LIN {X 0,Y 382.993,Z 296.779,A -85,B 0,C 180,E1 -12093.4,E2 -12093.4} C_VEL
LIN {X 0,Y 383.024,Z 296.771,A -85,B 0,C 180,E1 -12096.162,E2 -12096.162} C_VEL
LIN {X 0,Y 382.969,Z 296.778,A -85,B 0,C 180,E1 -12099.961,E2 -12099.961} C_VEL
LIN {X 0,Y 382.998,Z 296.778,A -85,B 0,C 180,E1 -12102.777,E2 -12102.777} C_VEL
LIN {X 0,Y 382.989,Z 296.776,A -85,B 0,C 180,E1 -12105.788,E2 -12105.788} C_VEL
LIN {X 0,Y 382.981,Z 296.782,A -85,B 0,C 180,E1 -12108.794,E2 -12108.794} C_VEL
LIN {X 0,Y 382.993,Z 296.776,A -85,B 0,C 180,E1 -12112.095,E2 -12112.095} C_VEL
LIN {X 0,Y 383.009,Z 296.776,A -85,B 0,C 180,E1 -12115.331,E2 -12115.331} C_VEL
LIN {X 0,Y 382.978,Z 296.781,A -85,B 0,C 180,E1 -12119.081,E2 -12119.081} C_VEL
LIN {X 0,Y 383.046,Z 296.772,A -85,B 0,C 180,E1 -12122.697,E2 -12122.697} C_VEL
LIN {X 0,Y 383.041,Z 296.772,A -85,B 0,C 180,E1 -12125.039,E2 -12125.039} C_VEL
LIN {X 0,Y 382.982,Z 296.78,A -85,B 0,C 180,E1 -12128.468,E2 -12128.468} C_VEL
LIN {X 0,Y 383.078,Z 296.767,A -85,B 0,C 180,E1 -12131.827,E2 -12131.827} C_VEL
LIN {X 0,Y 383.098,Z 296.763,A -85,B 0,C 180,E1 -12135.118,E2 -12135.118} C_VEL
LIN {X 0,Y 383.085,Z 296.769,A -85,B 0,C 180,E1 -12138.357,E2 -12138.357} C_VEL
LIN {X 0,Y 383.202,Z 296.753,A -85,B 0,C 180,E1 -12142.028,E2 -12142.028} C_VEL
LIN {X 0,Y 383.168,Z 296.754,A -85,B 0,C 180,E1 -12144.738,E2 -12144.738} C_VEL
LIN {X 0,Y 383.361,Z 296.733,A -85,B 0,C 180,E1 -12147.899,E2 -12147.899} C_VEL
LIN {X 0,Y 383.246,Z 296.743,A -85,B 0,C 180,E1 -12151.051,E2 -12151.051} C_VEL
LIN {X 0,Y 383.361,Z 296.733,A -85,B 0,C 180,E1 -12152.101,E2 -12152.101} C_VEL
LIN {X 0,Y 383.23,Z 296.747,A -85,B 0,C 180,E1 -12156.317,E2 -12156.317} C_VEL
LIN {X 0,Y 383.131,Z 296.762,A -85,B 0,C 180,E1 -12159.503,E2 -12159.503} C_VEL
LIN {X 0,Y 383.113,Z 296.766,A -85,B 0,C 180,E1 -12163.537,E2 -12163.537} C_VEL
LIN {X 0,Y 383.083,Z 296.769,A -85,B 0,C 180,E1 -12167.455,E2 -12167.455} C_VEL
LIN {X 0,Y 383.017,Z 296.773,A -85,B 0,C 180,E1 -12170.648,E2 -12170.648} C_VEL
LIN {X 0,Y 383.022,Z 296.775,A -85,B 0,C 180,E1 -12173.808,E2 -12173.808} C_VEL
LIN {X 0,Y 383.069,Z 296.767,A -85,B 0,C 180,E1 -12176.124,E2 -12176.124} C_VEL
LIN {X 0,Y 383.039,Z 296.771,A -85,B 0,C 180,E1 -12178.493,E2 -12178.493} C_VEL
LIN {X 0,Y 383.003,Z 296.775,A -85,B 0,C 180,E1 -12182.15,E2 -12182.15} C_VEL
LIN {X 0,Y 383.007,Z 296.775,A -85,B 0,C 180,E1 -12184.534,E2 -12184.534} C_VEL
LIN {X 0,Y 382.344,Z 296.861,A -85,B 0,C 180,E1 -12185.411,E2 -12185.411} C_VEL
LIN {X 0,Y 379.471,Z 297.217,A -85,B 0,C 180,E1 -12186.835,E2 -12186.835} C_VEL
LIN {X 0,Y 377.045,Z 297.517,A -85,B 0,C 180,E1 -12187.987,E2 -12187.987} C_VEL
LIN {X 0,Y 376.019,Z 297.647,A -85,B 0,C 180,E1 -12188.878,E2 -12188.878} C_VEL
LIN {X 0,Y 375.944,Z 297.654,A -85,B 0,C 180,E1 -12189.18,E2 -12189.18} C_VEL
LIN {X 0,Y 375.924,Z 297.657,A -85,B 0,C 180,E1 -12192.302,E2 -12192.302} C_VEL
LIN {X 0,Y 375.919,Z 297.66,A -85,B 0,C 180,E1 -12195.27,E2 -12195.27} C_VEL
LIN {X 0,Y 375.911,Z 297.659,A -85,B 0,C 180,E1 -12198.404,E2 -12198.404} C_VEL
LIN {X 0,Y 375.947,Z 297.652,A -85,B 0,C 180,E1 -12201.912,E2 -12201.912} C_VEL
LIN {X 0,Y 375.973,Z 297.65,A -85,B 0,C 180,E1 -12205.335,E2 -12205.335} C_VEL
LIN {X 0,Y 376.132,Z 297.715,A -85,B 0,C 180,E1 -12208.895,E2 -12208.895} C_VEL
LIN {X 0,Y 376.163,Z 302.091,A -85,B 0,C 180,E1 -12211.417,E2 -12211.417} C_VEL
LIN {X 0,Y 375.789,Z 308.656,A -85,B 0,C 180,E1 -12215.117,E2 -12215.117} C_VEL
LIN {X 0,Y 375.538,Z 314.97,A -85,B 0,C 180,E1 -12218.598,E2 -12218.598} C_VEL
LIN {X 0,Y 375.35,Z 320.211,A -85,B 0,C 180,E1 -12221.441,E2 -12221.441} C_VEL
LIN {X 0,Y 375.145,Z 326.489,A -85,B 0,C 180,E1 -12224.796,E2 -12224.796} C_VEL
LIN {X 0,Y 375.052,Z 332.791,A -85,B 0,C 180,E1 -12228.106,E2 -12228.106} C_VEL
LIN {X 0,Y 375.004,Z 334.24,A -85,B 0,C 180,E1 -12228.858,E2 -12228.858} C_VEL
LIN {X 0,Y 376.479,Z 346.042,A -85,B 0,C 180,E1 -12229.583,E2 -12229.583} C_VEL
LIN {X 0,Y 376.877,Z 352.36,A -85,B 0,C 180,E1 -12230.069,E2 -12230.069} C_VEL
LIN {X 0,Y 376.461,Z 362.339,A -85,B 0,C 180,E1 -12231.006,E2 -12231.006} C_VEL
LIN {X 0,Y 376.1,Z 370.955,A -85,B 0,C 180,E1 -12232.05,E2 -12232.05} C_VEL
LIN {X 0,Y 375.834,Z 378.97,A -85,B 0,C 180,E1 -12233.29,E2 -12233.29} C_VEL
LIN {X 0,Y 375.594,Z 385.708,A -85,B 0,C 180,E1 -12234.633,E2 -12234.633} C_VEL
LIN {X 0,Y 375.366,Z 389.937,A -85,B 0,C 180,E1 -12235.706,E2 -12235.706} C_VEL
LIN {X 0,Y 375.173,Z 393.311,A -85,B 0,C 180,E1 -12236.78,E2 -12236.78} C_VEL
LIN {X 0,Y 375.035,Z 395.913,A -85,B 0,C 180,E1 -12237.854,E2 -12237.854} C_VEL
LIN {X 0,Y 374.985,Z 397.794,A -85,B 0,C 180,E1 -12238.928,E2 -12238.928} C_VEL
LIN {X 0,Y 374.972,Z 398.993,A -85,B 0,C 180,E1 -12240.001,E2 -12240.001} C_VEL
LIN {X 0,Y 375.035,Z 399.523,A -85,B 0,C 180,E1 -12241.075,E2 -12241.075} C_VEL
LIN {X 0,Y 375.176,Z 399.397,A -85,B 0,C 180,E1 -12242.148,E2 -12242.148} C_VEL
LIN {X 0,Y 375.419,Z 398.616,A -85,B 0,C 180,E1 -12243.221,E2 -12243.221} C_VEL
LIN {X 0,Y 376.126,Z 396.159,A -85,B 0,C 180,E1 -12244.825,E2 -12244.825} C_VEL
LIN {X 0,Y 376.703,Z 392.135,A -85,B 0,C 180,E1 -12246.428,E2 -12246.428} C_VEL
LIN {X 0,Y 377.569,Z 386.275,A -85,B 0,C 180,E1 -12248.026,E2 -12248.026} C_VEL
LIN {X 0,Y 378.359,Z 379.801,A -85,B 0,C 180,E1 -12249.355,E2 -12249.355} C_VEL
LIN {X 0,Y 379.334,Z 372.3,A -85,B 0,C 180,E1 -12250.549,E2 -12250.549} C_VEL
LIN {X 0,Y 380.313,Z 362.823,A -85,B 0,C 180,E1 -12251.73,E2 -12251.73} C_VEL
LIN {X 0,Y 380.625,Z 357.706,A -85,B 0,C 180,E1 -12252.261,E2 -12252.261} C_VEL
LIN {X 0,Y 379.01,Z 348.75,A -85,B 0,C 180,E1 -12253.193,E2 -12253.193} C_VEL
LIN {X 0,Y 376.292,Z 338.883,A -85,B 0,C 180,E1 -12254.122,E2 -12254.122} C_VEL
LIN {X 0,Y 376.791,Z 332.831,A -85,B 0,C 180,E1 -12257.96,E2 -12257.96} C_VEL
LIN {X 0,Y 377.374,Z 327.03,A -85,B 0,C 180,E1 -12261.869,E2 -12261.869} C_VEL
LIN {X 0,Y 377.99,Z 322.325,A -85,B 0,C 180,E1 -12265.319,E2 -12265.319} C_VEL
LIN {X 0,Y 378.845,Z 317.93,A -85,B 0,C 180,E1 -12268.839,E2 -12268.839} C_VEL
LIN {X 0,Y 379.207,Z 315.14,A -85,B 0,C 180,E1 -12271.511,E2 -12271.511} C_VEL
LIN {X 0,Y 379.155,Z 313.11,A -85,B 0,C 180,E1 -12273.786,E2 -12273.786} C_VEL
LIN {X 0,Y 379.022,Z 311.404,A -85,B 0,C 180,E1 -12276.397,E2 -12276.397} C_VEL
LIN {X 0,Y 378.859,Z 310.258,A -85,B 0,C 180,E1 -12279.104,E2 -12279.104} C_VEL
LIN {X 0,Y 378.886,Z 309.796,A -85,B 0,C 180,E1 -12282.101,E2 -12282.101} C_VEL
LIN {X 0,Y 379.077,Z 310.446,A -85,B 0,C 180,E1 -12285.21,E2 -12285.21} C_VEL
LIN {X 0,Y 379.596,Z 312.145,A -85,B 0,C 180,E1 -12288.201,E2 -12288.201} C_VEL
LIN {X 0,Y 380.322,Z 314.889,A -85,B 0,C 180,E1 -12291.076,E2 -12291.076} C_VEL
LIN {X 0,Y 381.298,Z 319.139,A -85,B 0,C 180,E1 -12294.195,E2 -12294.195} C_VEL
LIN {X 0,Y 382.493,Z 324.452,A -85,B 0,C 180,E1 -12297.178,E2 -12297.178} C_VEL
LIN {X 0,Y 383.114,Z 328.518,A -85,B 0,C 180,E1 -12299.093,E2 -12299.093} C_VEL
LIN {X 0,Y 382.773,Z 331.551,A -85,B 0,C 180,E1 -12300.281,E2 -12300.281} C_VEL
LIN {X 0,Y 380.4,Z 341.516,A -85,B 0,C 180,E1 -12303.678,E2 -12303.678} C_VEL
LIN {X 0,Y 378.337,Z 354.145,A -85,B 0,C 180,E1 -12307.616,E2 -12307.616} C_VEL
LIN {X 0,Y 377.129,Z 364.425,A -85,B 0,C 180,E1 -12310.537,E2 -12310.537} C_VEL
LIN {X 0,Y 379.386,Z 377.001,A -85,B 0,C 180,E1 -12311.197,E2 -12311.197} C_VEL
LIN {X 0,Y 380.292,Z 388.82,A -85,B 0,C 180,E1 -12311.915,E2 -12311.915} C_VEL
LIN {X 0,Y 380.196,Z 399.286,A -85,B 0,C 180,E1 -12312.67,E2 -12312.67} C_VEL
LIN {X 0,Y 379.013,Z 411.289,A -85,B 0,C 180,E1 -12313.712,E2 -12313.712} C_VEL
LIN {X 0,Y 377.852,Z 422.147,A -85,B 0,C 180,E1 -12314.906,E2 -12314.906} C_VEL
LIN {X 0,Y 376.925,Z 431.899,A -85,B 0,C 180,E1 -12316.247,E2 -12316.247} C_VEL
LIN {X 0,Y 376.109,Z 439.941,A -85,B 0,C 180,E1 -12317.591,E2 -12317.591} C_VEL
LIN {X 0,Y 375.361,Z 447.84,A -85,B 0,C 180,E1 -12319.209,E2 -12319.209} C_VEL
LIN {X 0,Y 374.984,Z 454.183,A -85,B 0,C 180,E1 -12320.833,E2 -12320.833} C_VEL
LIN {X 0,Y 374.858,Z 459.235,A -85,B 0,C 180,E1 -12322.459,E2 -12322.459} C_VEL
LIN {X 0,Y 374.782,Z 462.239,A -85,B 0,C 180,E1 -12323.659,E2 -12323.659} C_VEL
LIN {X 0,Y 374.773,Z 464.187,A -85,B 0,C 180,E1 -12324.62,E2 -12324.62} C_VEL
LIN {X 0,Y 374.759,Z 465.952,A -85,B 0,C 180,E1 -12325.698,E2 -12325.698} C_VEL
LIN {X 0,Y 374.922,Z 467.299,A -85,B 0,C 180,E1 -12326.776,E2 -12326.776} C_VEL
LIN {X 0,Y 374.99,Z 468.16,A -85,B 0,C 180,E1 -12327.852,E2 -12327.852} C_VEL
LIN {X 0,Y 374.931,Z 468.593,A -85,B 0,C 180,E1 -12328.926,E2 -12328.926} C_VEL
LIN {X 0,Y 374.902,Z 468.611,A -85,B 0,C 180,E1 -12330,E2 -12330} C_VEL
LIN {X 0,Y 374.93,Z 468.155,A -85,B 0,C 180,E1 -12331.074,E2 -12331.074} C_VEL
LIN {X 0,Y 375.039,Z 467.282,A -85,B 0,C 180,E1 -12332.148,E2 -12332.148} C_VEL
LIN {X 0,Y 374.995,Z 465.962,A -85,B 0,C 180,E1 -12333.223,E2 -12333.223} C_VEL
LIN {X 0,Y 374.841,Z 463.042,A -85,B 0,C 180,E1 -12334.84,E2 -12334.84} C_VEL
LIN {X 0,Y 374.949,Z 458.664,A -85,B 0,C 180,E1 -12336.567,E2 -12336.567} C_VEL
LIN {X 0,Y 374.995,Z 452.62,A -85,B 0,C 180,E1 -12338.352,E2 -12338.352} C_VEL
LIN {X 0,Y 375.182,Z 445.526,A -85,B 0,C 180,E1 -12339.978,E2 -12339.978} C_VEL
LIN {X 0,Y 375.676,Z 436.584,A -85,B 0,C 180,E1 -12341.602,E2 -12341.602} C_VEL
LIN {X 0,Y 376.261,Z 427.274,A -85,B 0,C 180,E1 -12342.953,E2 -12342.953} C_VEL
LIN {X 0,Y 376.815,Z 416.818,A -85,B 0,C 180,E1 -12344.17,E2 -12344.17} C_VEL
LIN {X 0,Y 377.38,Z 406.757,A -85,B 0,C 180,E1 -12345.113,E2 -12345.113} C_VEL
LIN {X 0,Y 378.045,Z 394.838,A -85,B 0,C 180,E1 -12345.984,E2 -12345.984} C_VEL
LIN {X 0,Y 377.323,Z 383.251,A -85,B 0,C 180,E1 -12346.641,E2 -12346.641} C_VEL
LIN {X 0,Y 376.34,Z 371.136,A -85,B 0,C 180,E1 -12347.14,E2 -12347.14} C_VEL
LIN {X 0,Y 376.014,Z 366.072,A -85,B 0,C 180,E1 -12347.296,E2 -12347.296} C_VEL
LIN {X 0,Y 377.114,Z 351.417,A -85,B 0,C 180,E1 -12351.278,E2 -12351.278} C_VEL
LIN {X 0,Y 378.263,Z 339.903,A -85,B 0,C 180,E1 -12354.437,E2 -12354.437} C_VEL
LIN {X 0,Y 379.811,Z 327.577,A -85,B 0,C 180,E1 -12357.854,E2 -12357.854} C_VEL
LIN {X 0,Y 380.623,Z 320.323,A -85,B 0,C 180,E1 -12359.904,E2 -12359.904} C_VEL
LIN {X 0,Y 378.647,Z 310.587,A -85,B 0,C 180,E1 -12362.917,E2 -12362.917} C_VEL
LIN {X 0,Y 376.227,Z 298.875,A -85,B 0,C 180,E1 -12366.71,E2 -12366.71} C_VEL
LIN {X 0,Y 375.972,Z 297.654,A -85,B 0,C 180,E1 -12367.158,E2 -12367.158} C_VEL
LIN {X 0,Y 375.945,Z 297.656,A -85,B 0,C 180,E1 -12370.867,E2 -12370.867} C_VEL
LIN {X 0,Y 375.935,Z 297.658,A -85,B 0,C 180,E1 -12373.765,E2 -12373.765} C_VEL
LIN {X 0,Y 375.939,Z 297.655,A -85,B 0,C 180,E1 -12376.81,E2 -12376.81} C_VEL
LIN {X 0,Y 375.968,Z 297.655,A -85,B 0,C 180,E1 -12380.537,E2 -12380.537} C_VEL
LIN {X 0,Y 375.969,Z 297.655,A -85,B 0,C 180,E1 -12383.495,E2 -12383.495} C_VEL
LIN {X 0,Y 375.969,Z 297.686,A -85,B 0,C 180,E1 -12385.888,E2 -12385.888} C_VEL
LIN {X 0,Y 377.371,Z 303.877,A -85,B 0,C 180,E1 -12388.947,E2 -12388.947} C_VEL
LIN {X 0,Y 377.839,Z 308.436,A -85,B 0,C 180,E1 -12391.077,E2 -12391.077} C_VEL
LIN {X 0,Y 377.468,Z 316.369,A -85,B 0,C 180,E1 -12394.643,E2 -12394.643} C_VEL
LIN {X 0,Y 377.21,Z 324.059,A -85,B 0,C 180,E1 -12398.121,E2 -12398.121} C_VEL
LIN {X 0,Y 376.985,Z 331.514,A -85,B 0,C 180,E1 -12401.522,E2 -12401.522} C_VEL
LIN {X 0,Y 376.762,Z 338.786,A -85,B 0,C 180,E1 -12404.86,E2 -12404.86} C_VEL
LIN {X 0,Y 376.729,Z 345.225,A -85,B 0,C 180,E1 -12407.764,E2 -12407.764} C_VEL
LIN {X 0,Y 379.03,Z 354.751,A -85,B 0,C 180,E1 -12408.501,E2 -12408.501} C_VEL
LIN {X 0,Y 379.112,Z 359.76,A -85,B 0,C 180,E1 -12408.91,E2 -12408.91} C_VEL
LIN {X 0,Y 378.621,Z 367.683,A -85,B 0,C 180,E1 -12409.672,E2 -12409.672} C_VEL
LIN {X 0,Y 377.863,Z 375.923,A -85,B 0,C 180,E1 -12410.705,E2 -12410.705} C_VEL
LIN {X 0,Y 377.418,Z 382.05,A -85,B 0,C 180,E1 -12411.701,E2 -12411.701} C_VEL
LIN {X 0,Y 376.994,Z 387.186,A -85,B 0,C 180,E1 -12412.77,E2 -12412.77} C_VEL
LIN {X 0,Y 376.468,Z 392.079,A -85,B 0,C 180,E1 -12414.105,E2 -12414.105} C_VEL
LIN {X 0,Y 376.109,Z 394.999,A -85,B 0,C 180,E1 -12415.175,E2 -12415.175} C_VEL
LIN {X 0,Y 375.379,Z 397.85,A -85,B 0,C 180,E1 -12416.779,E2 -12416.779} C_VEL
LIN {X 0,Y 375.142,Z 398.857,A -85,B 0,C 180,E1 -12417.851,E2 -12417.851} C_VEL
LIN {X 0,Y 375.01,Z 399.169,A -85,B 0,C 180,E1 -12418.925,E2 -12418.925} C_VEL
LIN {X 0,Y 374.955,Z 398.796,A -85,B 0,C 180,E1 -12419.999,E2 -12419.999} C_VEL
LIN {X 0,Y 374.976,Z 397.723,A -85,B 0,C 180,E1 -12421.073,E2 -12421.073} C_VEL
LIN {X 0,Y 375.035,Z 395.927,A -85,B 0,C 180,E1 -12422.146,E2 -12422.146} C_VEL
LIN {X 0,Y 375.309,Z 391.751,A -85,B 0,C 180,E1 -12423.756,E2 -12423.756} C_VEL
LIN {X 0,Y 375.545,Z 386.75,A -85,B 0,C 180,E1 -12425.098,E2 -12425.098} C_VEL
LIN {X 0,Y 375.658,Z 381.546,A -85,B 0,C 180,E1 -12426.174,E2 -12426.174} C_VEL
LIN {X 0,Y 375.825,Z 374.325,A -85,B 0,C 180,E1 -12427.337,E2 -12427.337} C_VEL
LIN {X 0,Y 376.022,Z 366.64,A -85,B 0,C 180,E1 -12428.3,E2 -12428.3} C_VEL
LIN {X 0,Y 376.267,Z 357.879,A -85,B 0,C 180,E1 -12429.134,E2 -12429.134} C_VEL
LIN {X 0,Y 376.381,Z 348.482,A -85,B 0,C 180,E1 -12429.809,E2 -12429.809} C_VEL
LIN {X 0,Y 375.44,Z 341.359,A -85,B 0,C 180,E1 -12430.208,E2 -12430.208} C_VEL
LIN {X 0,Y 375.56,Z 334.224,A -85,B 0,C 180,E1 -12433.319,E2 -12433.319} C_VEL
LIN {X 0,Y 375.568,Z 325.063,A -85,B 0,C 180,E1 -12437.376,E2 -12437.376} C_VEL
LIN {X 0,Y 375.686,Z 317.354,A -85,B 0,C 180,E1 -12440.818,E2 -12440.818} C_VEL
LIN {X 0,Y 375.83,Z 309.622,A -85,B 0,C 180,E1 -12444.291,E2 -12444.291} C_VEL
LIN {X 0,Y 375.918,Z 303.002,A -85,B 0,C 180,E1 -12447.259,E2 -12447.259} C_VEL
LIN {X 0,Y 376.07,Z 297.64,A -85,B 0,C 180,E1 -12449.683,E2 -12449.683} C_VEL
LIN {X 0,Y 375.942,Z 297.655,A -85,B 0,C 180,E1 -12452.827,E2 -12452.827} C_VEL
LIN {X 0,Y 375.95,Z 297.656,A -85,B 0,C 180,E1 -12455.414,E2 -12455.414} C_VEL
LIN {X 0,Y 375.93,Z 297.655,A -85,B 0,C 180,E1 -12458.262,E2 -12458.262} C_VEL
LIN {X 0,Y 375.912,Z 297.659,A -85,B 0,C 180,E1 -12461.597,E2 -12461.597} C_VEL
LIN {X 0,Y 375.919,Z 297.66,A -85,B 0,C 180,E1 -12464.73,E2 -12464.73} C_VEL
LIN {X 0,Y 375.927,Z 297.657,A -85,B 0,C 180,E1 -12468.398,E2 -12468.398} C_VEL
LIN {X 0,Y 375.968,Z 297.651,A -85,B 0,C 180,E1 -12471.728,E2 -12471.728} C_VEL
LIN {X 0,Y 375.971,Z 297.652,A -85,B 0,C 180,E1 -12475.331,E2 -12475.331} C_VEL
LIN {X 0,Y 375.952,Z 297.657,A -85,B 0,C 180,E1 -12478.437,E2 -12478.437} C_VEL
LIN {X 0,Y 375.992,Z 297.65,A -85,B 0,C 180,E1 -12482.141,E2 -12482.141} C_VEL
LIN {X 0,Y 375.996,Z 297.651,A -85,B 0,C 180,E1 -12484.538,E2 -12484.538} C_VEL
LIN {X 0,Y 375.952,Z 297.655,A -85,B 0,C 180,E1 -12488.045,E2 -12488.045} C_VEL
LIN {X 0,Y 376.012,Z 297.645,A -85,B 0,C 180,E1 -12491.473,E2 -12491.473} C_VEL
LIN {X 0,Y 376.046,Z 297.643,A -85,B 0,C 180,E1 -12494.832,E2 -12494.832} C_VEL
LIN {X 0,Y 376.037,Z 297.645,A -85,B 0,C 180,E1 -12498.136,E2 -12498.136} C_VEL
LIN {X 0,Y 376.174,Z 297.628,A -85,B 0,C 180,E1 -12501.953,E2 -12501.953} C_VEL
LIN {X 0,Y 376.139,Z 297.63,A -85,B 0,C 180,E1 -12504.639,E2 -12504.639} C_VEL
LIN {X 0,Y 376.325,Z 297.609,A -85,B 0,C 180,E1 -12507.859,E2 -12507.859} C_VEL
LIN {X 0,Y 376.218,Z 297.618,A -85,B 0,C 180,E1 -12511.07,E2 -12511.07} C_VEL
LIN {X 0,Y 376.326,Z 297.609,A -85,B 0,C 180,E1 -12512.141,E2 -12512.141} C_VEL
LIN {X 0,Y 376.189,Z 297.624,A -85,B 0,C 180,E1 -12516.436,E2 -12516.436} C_VEL
LIN {X 0,Y 376.101,Z 297.639,A -85,B 0,C 180,E1 -12519.682,E2 -12519.682} C_VEL
LIN {X 0,Y 376.077,Z 297.641,A -85,B 0,C 180,E1 -12523.658,E2 -12523.658} C_VEL
LIN {X 0,Y 376.033,Z 297.646,A -85,B 0,C 180,E1 -12527.608,E2 -12527.608} C_VEL
LIN {X 0,Y 375.967,Z 297.652,A -85,B 0,C 180,E1 -12530.833,E2 -12530.833} C_VEL
LIN {X 0,Y 375.983,Z 297.649,A -85,B 0,C 180,E1 -12534.282,E2 -12534.282} C_VEL
LIN {X 0,Y 376.009,Z 297.646,A -85,B 0,C 180,E1 -12536.653,E2 -12536.653} C_VEL
LIN {X 0,Y 375.967,Z 297.655,A -85,B 0,C 180,E1 -12539.08,E2 -12539.08} C_VEL
LIN {X 0,Y 375.941,Z 297.657,A -85,B 0,C 180,E1 -12542.83,E2 -12542.83} C_VEL
LIN {X 0,Y 375.949,Z 297.657,A -85,B 0,C 180,E1 -12545.417,E2 -12545.417} C_VEL
LIN {X 0,Y 375.944,Z 297.654,A -85,B 0,C 180,E1 -12549.18,E2 -12549.18} C_VEL
LIN {X 0,Y 375.299,Z 297.739,A -85,B 0,C 180,E1 -12550.074,E2 -12550.074} C_VEL
LIN {X 0,Y 372.447,Z 298.096,A -85,B 0,C 180,E1 -12551.527,E2 -12551.527} C_VEL
LIN {X 0,Y 370.01,Z 298.396,A -85,B 0,C 180,E1 -12552.702,E2 -12552.702} C_VEL
LIN {X 0,Y 368.951,Z 298.526,A -85,B 0,C 180,E1 -12553.611,E2 -12553.611} C_VEL
LIN {X 0,Y 368.859,Z 298.536,A -85,B 0,C 180,E1 -12553.919,E2 -12553.919} C_VEL
LIN {X 0,Y 368.878,Z 298.536,A -85,B 0,C 180,E1 -12556.697,E2 -12556.697} C_VEL
LIN {X 0,Y 368.877,Z 298.534,A -85,B 0,C 180,E1 -12559.65,E2 -12559.65} C_VEL
LIN {X 0,Y 368.893,Z 298.534,A -85,B 0,C 180,E1 -12563.146,E2 -12563.146} C_VEL
LIN {X 0,Y 368.897,Z 298.534,A -85,B 0,C 180,E1 -12566.464,E2 -12566.464} C_VEL
LIN {X 0,Y 369.102,Z 298.71,A -85,B 0,C 180,E1 -12568.9,E2 -12568.9} C_VEL
LIN {X 0,Y 369.151,Z 302.525,A -85,B 0,C 180,E1 -12571.136,E2 -12571.136} C_VEL
LIN {X 0,Y 368.741,Z 309.691,A -85,B 0,C 180,E1 -12575.211,E2 -12575.211} C_VEL
LIN {X 0,Y 368.49,Z 316.032,A -85,B 0,C 180,E1 -12578.756,E2 -12578.756} C_VEL
LIN {X 0,Y 368.241,Z 322.345,A -85,B 0,C 180,E1 -12582.222,E2 -12582.222} C_VEL
LIN {X 0,Y 368.028,Z 328.681,A -85,B 0,C 180,E1 -12585.627,E2 -12585.627} C_VEL
LIN {X 0,Y 367.96,Z 334.513,A -85,B 0,C 180,E1 -12588.712,E2 -12588.712} C_VEL
LIN {X 0,Y 369.359,Z 346.143,A -85,B 0,C 180,E1 -12589.449,E2 -12589.449} C_VEL
LIN {X 0,Y 369.864,Z 351.695,A -85,B 0,C 180,E1 -12589.878,E2 -12589.878} C_VEL
LIN {X 0,Y 369.427,Z 361.928,A -85,B 0,C 180,E1 -12590.834,E2 -12590.834} C_VEL
LIN {X 0,Y 369.073,Z 370.367,A -85,B 0,C 180,E1 -12591.846,E2 -12591.846} C_VEL
LIN {X 0,Y 368.793,Z 378.958,A -85,B 0,C 180,E1 -12593.161,E2 -12593.161} C_VEL
LIN {X 0,Y 368.522,Z 385.864,A -85,B 0,C 180,E1 -12594.53,E2 -12594.53} C_VEL
LIN {X 0,Y 368.293,Z 390.223,A -85,B 0,C 180,E1 -12595.624,E2 -12595.624} C_VEL
LIN {X 0,Y 368.119,Z 393.693,A -85,B 0,C 180,E1 -12596.718,E2 -12596.718} C_VEL
LIN {X 0,Y 367.963,Z 396.376,A -85,B 0,C 180,E1 -12597.812,E2 -12597.812} C_VEL
LIN {X 0,Y 367.934,Z 398.338,A -85,B 0,C 180,E1 -12598.907,E2 -12598.907} C_VEL
LIN {X 0,Y 367.918,Z 399.628,A -85,B 0,C 180,E1 -12600.001,E2 -12600.001} C_VEL
LIN {X 0,Y 367.983,Z 400.258,A -85,B 0,C 180,E1 -12601.096,E2 -12601.096} C_VEL
LIN {X 0,Y 368.131,Z 400.226,A -85,B 0,C 180,E1 -12602.19,E2 -12602.19} C_VEL
LIN {X 0,Y 368.391,Z 399.532,A -85,B 0,C 180,E1 -12603.282,E2 -12603.282} C_VEL
LIN {X 0,Y 369.127,Z 397.211,A -85,B 0,C 180,E1 -12604.916,E2 -12604.916} C_VEL
LIN {X 0,Y 369.754,Z 393.369,A -85,B 0,C 180,E1 -12606.55,E2 -12606.55} C_VEL
LIN {X 0,Y 370.694,Z 387.767,A -85,B 0,C 180,E1 -12608.176,E2 -12608.176} C_VEL
LIN {X 0,Y 371.536,Z 381.535,A -85,B 0,C 180,E1 -12609.528,E2 -12609.528} C_VEL
LIN {X 0,Y 372.653,Z 373.421,A -85,B 0,C 180,E1 -12610.872,E2 -12610.872} C_VEL
LIN {X 0,Y 373.711,Z 364.148,A -85,B 0,C 180,E1 -12612.064,E2 -12612.064} C_VEL
LIN {X 0,Y 374.024,Z 359.119,A -85,B 0,C 180,E1 -12612.618,E2 -12612.618} C_VEL
LIN {X 0,Y 372.318,Z 349.495,A -85,B 0,C 180,E1 -12613.678,E2 -12613.678} C_VEL
LIN {X 0,Y 369.384,Z 339.417,A -85,B 0,C 180,E1 -12614.691,E2 -12614.691} C_VEL
LIN {X 0,Y 369.865,Z 334.06,A -85,B 0,C 180,E1 -12618.18,E2 -12618.18} C_VEL
LIN {X 0,Y 370.538,Z 328.16,A -85,B 0,C 180,E1 -12622.294,E2 -12622.294} C_VEL
LIN {X 0,Y 371.228,Z 323.512,A -85,B 0,C 180,E1 -12625.814,E2 -12625.814} C_VEL
LIN {X 0,Y 372.163,Z 319.321,A -85,B 0,C 180,E1 -12629.407,E2 -12629.407} C_VEL
LIN {X 0,Y 372.402,Z 316.848,A -85,B 0,C 180,E1 -12631.9,E2 -12631.9} C_VEL
LIN {X 0,Y 372.394,Z 314.86,A -85,B 0,C 180,E1 -12634.485,E2 -12634.485} C_VEL
LIN {X 0,Y 372.239,Z 313.198,A -85,B 0,C 180,E1 -12637.535,E2 -12637.535} C_VEL
LIN {X 0,Y 372.164,Z 312.509,A -85,B 0,C 180,E1 -12639.947,E2 -12639.947} C_VEL
LIN {X 0,Y 372.274,Z 312.393,A -85,B 0,C 180,E1 -12642.816,E2 -12642.816} C_VEL
LIN {X 0,Y 372.524,Z 313.266,A -85,B 0,C 180,E1 -12645.801,E2 -12645.801} C_VEL
LIN {X 0,Y 373.083,Z 315.153,A -85,B 0,C 180,E1 -12648.752,E2 -12648.752} C_VEL
LIN {X 0,Y 373.803,Z 318.115,A -85,B 0,C 180,E1 -12651.651,E2 -12651.651} C_VEL
LIN {X 0,Y 374.727,Z 322.033,A -85,B 0,C 180,E1 -12654.45,E2 -12654.45} C_VEL
LIN {X 0,Y 375.851,Z 327.091,A -85,B 0,C 180,E1 -12657.295,E2 -12657.295} C_VEL
LIN {X 0,Y 376.354,Z 331.066,A -85,B 0,C 180,E1 -12659.206,E2 -12659.206} C_VEL
LIN {X 0,Y 375.395,Z 335.43,A -85,B 0,C 180,E1 -12660.872,E2 -12660.872} C_VEL
LIN {X 0,Y 373.067,Z 345.476,A -85,B 0,C 180,E1 -12664.324,E2 -12664.324} C_VEL
LIN {X 0,Y 371.072,Z 357.601,A -85,B 0,C 180,E1 -12668.135,E2 -12668.135} C_VEL
LIN {X 0,Y 370.306,Z 363.846,A -85,B 0,C 180,E1 -12669.988,E2 -12669.988} C_VEL
LIN {X 0,Y 372.821,Z 377.567,A -85,B 0,C 180,E1 -12670.762,E2 -12670.762} C_VEL
LIN {X 0,Y 373.693,Z 389.215,A -85,B 0,C 180,E1 -12671.517,E2 -12671.517} C_VEL
LIN {X 0,Y 373.491,Z 400.085,A -85,B 0,C 180,E1 -12672.343,E2 -12672.343} C_VEL
LIN {X 0,Y 372.225,Z 411.819,A -85,B 0,C 180,E1 -12673.407,E2 -12673.407} C_VEL
LIN {X 0,Y 371.016,Z 422.358,A -85,B 0,C 180,E1 -12674.621,E2 -12674.621} C_VEL
LIN {X 0,Y 370.003,Z 431.935,A -85,B 0,C 180,E1 -12675.985,E2 -12675.985} C_VEL
LIN {X 0,Y 369.152,Z 439.833,A -85,B 0,C 180,E1 -12677.353,E2 -12677.353} C_VEL
LIN {X 0,Y 368.352,Z 447.578,A -85,B 0,C 180,E1 -12679.001,E2 -12679.001} C_VEL
LIN {X 0,Y 367.931,Z 453.824,A -85,B 0,C 180,E1 -12680.656,E2 -12680.656} C_VEL
LIN {X 0,Y 367.758,Z 458.797,A -85,B 0,C 180,E1 -12682.312,E2 -12682.312} C_VEL
LIN {X 0,Y 367.703,Z 462.007,A -85,B 0,C 180,E1 -12683.67,E2 -12683.67} C_VEL
LIN {X 0,Y 367.679,Z 465.376,A -85,B 0,C 180,E1 -12685.615,E2 -12685.615} C_VEL
LIN {X 0,Y 367.835,Z 466.662,A -85,B 0,C 180,E1 -12686.714,E2 -12686.714} C_VEL
LIN {X 0,Y 367.912,Z 467.49,A -85,B 0,C 180,E1 -12687.81,E2 -12687.81} C_VEL
LIN {X 0,Y 367.884,Z 467.896,A -85,B 0,C 180,E1 -12688.905,E2 -12688.905} C_VEL
LIN {X 0,Y 367.852,Z 467.855,A -85,B 0,C 180,E1 -12690,E2 -12690} C_VEL
LIN {X 0,Y 367.884,Z 467.36,A -85,B 0,C 180,E1 -12691.095,E2 -12691.095} C_VEL
LIN {X 0,Y 367.991,Z 466.456,A -85,B 0,C 180,E1 -12692.189,E2 -12692.189} C_VEL
LIN {X 0,Y 367.929,Z 465.066,A -85,B 0,C 180,E1 -12693.285,E2 -12693.285} C_VEL
LIN {X 0,Y 367.785,Z 462.062,A -85,B 0,C 180,E1 -12694.933,E2 -12694.933} C_VEL
LIN {X 0,Y 367.886,Z 457.921,A -85,B 0,C 180,E1 -12696.582,E2 -12696.582} C_VEL
LIN {X 0,Y 367.905,Z 452.463,A -85,B 0,C 180,E1 -12698.237,E2 -12698.237} C_VEL
LIN {X 0,Y 368.088,Z 445.531,A -85,B 0,C 180,E1 -12699.895,E2 -12699.895} C_VEL
LIN {X 0,Y 368.566,Z 436.724,A -85,B 0,C 180,E1 -12701.55,E2 -12701.55} C_VEL
LIN {X 0,Y 369.11,Z 427.615,A -85,B 0,C 180,E1 -12702.928,E2 -12702.928} C_VEL
LIN {X 0,Y 369.668,Z 417.425,A -85,B 0,C 180,E1 -12704.162,E2 -12704.162} C_VEL
LIN {X 0,Y 370.348,Z 406.001,A -85,B 0,C 180,E1 -12705.266,E2 -12705.266} C_VEL
LIN {X 0,Y 370.973,Z 393.972,A -85,B 0,C 180,E1 -12706.156,E2 -12706.156} C_VEL
LIN {X 0,Y 370.123,Z 382.222,A -85,B 0,C 180,E1 -12706.832,E2 -12706.832} C_VEL
LIN {X 0,Y 369.2,Z 369.792,A -85,B 0,C 180,E1 -12707.339,E2 -12707.339} C_VEL
LIN {X 0,Y 368.967,Z 365.824,A -85,B 0,C 180,E1 -12707.458,E2 -12707.458} C_VEL
LIN {X 0,Y 370.105,Z 351.353,A -85,B 0,C 180,E1 -12711.49,E2 -12711.49} C_VEL
LIN {X 0,Y 371.309,Z 339.964,A -85,B 0,C 180,E1 -12714.695,E2 -12714.695} C_VEL
LIN {X 0,Y 372.873,Z 327.949,A -85,B 0,C 180,E1 -12718.113,E2 -12718.113} C_VEL
LIN {X 0,Y 373.594,Z 321.174,A -85,B 0,C 180,E1 -12720.076,E2 -12720.076} C_VEL
LIN {X 0,Y 371.292,Z 310.031,A -85,B 0,C 180,E1 -12723.605,E2 -12723.605} C_VEL
LIN {X 0,Y 369.083,Z 299.351,A -85,B 0,C 180,E1 -12727.168,E2 -12727.168} C_VEL
LIN {X 0,Y 368.932,Z 298.532,A -85,B 0,C 180,E1 -12727.466,E2 -12727.466} C_VEL
LIN {X 0,Y 368.916,Z 298.534,A -85,B 0,C 180,E1 -12730.37,E2 -12730.37} C_VEL
LIN {X 0,Y 368.888,Z 298.535,A -85,B 0,C 180,E1 -12733.615,E2 -12733.615} C_VEL
LIN {X 0,Y 368.891,Z 298.533,A -85,B 0,C 180,E1 -12736.695,E2 -12736.695} C_VEL
LIN {X 0,Y 368.917,Z 298.53,A -85,B 0,C 180,E1 -12739.642,E2 -12739.642} C_VEL
LIN {X 0,Y 368.907,Z 298.535,A -85,B 0,C 180,E1 -12743.144,E2 -12743.144} C_VEL
LIN {X 0,Y 368.959,Z 298.612,A -85,B 0,C 180,E1 -12744.992,E2 -12744.992} C_VEL
LIN {X 0,Y 370.252,Z 304.216,A -85,B 0,C 180,E1 -12747.893,E2 -12747.893} C_VEL
LIN {X 0,Y 370.993,Z 308.167,A -85,B 0,C 180,E1 -12749.866,E2 -12749.866} C_VEL
LIN {X 0,Y 371.039,Z 312.132,A -85,B 0,C 180,E1 -12751.735,E2 -12751.735} C_VEL
LIN {X 0,Y 370.582,Z 320.491,A -85,B 0,C 180,E1 -12755.549,E2 -12755.549} C_VEL
LIN {X 0,Y 370.278,Z 328.903,A -85,B 0,C 180,E1 -12759.442,E2 -12759.442} C_VEL
LIN {X 0,Y 369.997,Z 337.494,A -85,B 0,C 180,E1 -12763.445,E2 -12763.445} C_VEL
LIN {X 0,Y 369.813,Z 345.979,A -85,B 0,C 180,E1 -12767.357,E2 -12767.357} C_VEL
LIN {X 0,Y 371.951,Z 354.234,A -85,B 0,C 180,E1 -12768.003,E2 -12768.003} C_VEL
LIN {X 0,Y 372.551,Z 357.54,A -85,B 0,C 180,E1 -12768.298,E2 -12768.298} C_VEL
LIN {X 0,Y 372.068,Z 366.434,A -85,B 0,C 180,E1 -12769.111,E2 -12769.111} C_VEL
LIN {X 0,Y 371.424,Z 374.088,A -85,B 0,C 180,E1 -12770.014,E2 -12770.014} C_VEL
LIN {X 0,Y 370.731,Z 381.043,A -85,B 0,C 180,E1 -12771.088,E2 -12771.088} C_VEL
LIN {X 0,Y 370.168,Z 387.39,A -85,B 0,C 180,E1 -12772.361,E2 -12772.361} C_VEL
LIN {X 0,Y 369.64,Z 391.528,A -85,B 0,C 180,E1 -12773.448,E2 -12773.448} C_VEL
LIN {X 0,Y 369.208,Z 394.736,A -85,B 0,C 180,E1 -12774.537,E2 -12774.537} C_VEL
LIN {X 0,Y 368.772,Z 397.133,A -85,B 0,C 180,E1 -12775.627,E2 -12775.627} C_VEL
LIN {X 0,Y 368.352,Z 398.78,A -85,B 0,C 180,E1 -12776.717,E2 -12776.717} C_VEL
LIN {X 0,Y 368.098,Z 399.701,A -85,B 0,C 180,E1 -12777.81,E2 -12777.81} C_VEL
LIN {X 0,Y 367.959,Z 399.919,A -85,B 0,C 180,E1 -12778.904,E2 -12778.904} C_VEL
LIN {X 0,Y 367.902,Z 399.439,A -85,B 0,C 180,E1 -12779.999,E2 -12779.999} C_VEL
LIN {X 0,Y 367.925,Z 398.258,A -85,B 0,C 180,E1 -12781.093,E2 -12781.093} C_VEL
LIN {X 0,Y 368.024,Z 395.114,A -85,B 0,C 180,E1 -12782.735,E2 -12782.735} C_VEL
LIN {X 0,Y 368.243,Z 392.067,A -85,B 0,C 180,E1 -12783.829,E2 -12783.829} C_VEL
LIN {X 0,Y 368.46,Z 386.888,A -85,B 0,C 180,E1 -12785.197,E2 -12785.197} C_VEL
LIN {X 0,Y 368.613,Z 381.567,A -85,B 0,C 180,E1 -12786.292,E2 -12786.292} C_VEL
LIN {X 0,Y 368.769,Z 374.08,A -85,B 0,C 180,E1 -12787.478,E2 -12787.478} C_VEL
LIN {X 0,Y 368.986,Z 365.895,A -85,B 0,C 180,E1 -12788.487,E2 -12788.487} C_VEL
LIN {X 0,Y 369.242,Z 357.014,A -85,B 0,C 180,E1 -12789.309,E2 -12789.309} C_VEL
LIN {X 0,Y 369.342,Z 349.316,A -85,B 0,C 180,E1 -12789.859,E2 -12789.859} C_VEL
LIN {X 0,Y 368.387,Z 341.906,A -85,B 0,C 180,E1 -12790.301,E2 -12790.301} C_VEL
LIN {X 0,Y 368.481,Z 333.928,A -85,B 0,C 180,E1 -12793.796,E2 -12793.796} C_VEL
LIN {X 0,Y 368.511,Z 325.546,A -85,B 0,C 180,E1 -12797.528,E2 -12797.528} C_VEL
LIN {X 0,Y 368.629,Z 318.017,A -85,B 0,C 180,E1 -12800.901,E2 -12800.901} C_VEL
LIN {X 0,Y 368.772,Z 309.429,A -85,B 0,C 180,E1 -12804.787,E2 -12804.787} C_VEL
LIN {X 0,Y 368.876,Z 302.599,A -85,B 0,C 180,E1 -12807.824,E2 -12807.824} C_VEL
LIN {X 0,Y 369.018,Z 298.518,A -85,B 0,C 180,E1 -12809.758,E2 -12809.758} C_VEL
LIN {X 0,Y 368.89,Z 298.534,A -85,B 0,C 180,E1 -12813.537,E2 -12813.537} C_VEL
LIN {X 0,Y 368.893,Z 298.534,A -85,B 0,C 180,E1 -12816.854,E2 -12816.854} C_VEL
LIN {X 0,Y 368.877,Z 298.534,A -85,B 0,C 180,E1 -12820.372,E2 -12820.372} C_VEL
LIN {X 0,Y 368.875,Z 298.535,A -85,B 0,C 180,E1 -12823.614,E2 -12823.614} C_VEL
LIN {X 0,Y 368.878,Z 298.537,A -85,B 0,C 180,E1 -12826.694,E2 -12826.694} C_VEL
LIN {X 0,Y 368.904,Z 298.531,A -85,B 0,C 180,E1 -12829.642,E2 -12829.642} C_VEL
LIN {X 0,Y 368.894,Z 298.535,A -85,B 0,C 180,E1 -12833.143,E2 -12833.143} C_VEL
LIN {X 0,Y 368.887,Z 298.536,A -85,B 0,C 180,E1 -12836.461,E2 -12836.461} C_VEL
LIN {X 0,Y 368.914,Z 298.532,A -85,B 0,C 180,E1 -12840.309,E2 -12840.309} C_VEL
LIN {X 0,Y 368.971,Z 298.522,A -85,B 0,C 180,E1 -12843.534,E2 -12843.534} C_VEL
LIN {X 0,Y 368.956,Z 298.528,A -85,B 0,C 180,E1 -12846.421,E2 -12846.421} C_VEL
LIN {X 0,Y 368.925,Z 298.53,A -85,B 0,C 180,E1 -12849.946,E2 -12849.946} C_VEL
LIN {X 0,Y 368.964,Z 298.523,A -85,B 0,C 180,E1 -12853.398,E2 -12853.398} C_VEL
LIN {X 0,Y 369.046,Z 298.514,A -85,B 0,C 180,E1 -12856.79,E2 -12856.79} C_VEL
LIN {X 0,Y 369.051,Z 298.516,A -85,B 0,C 180,E1 -12860.131,E2 -12860.131} C_VEL
LIN {X 0,Y 369.149,Z 298.5,A -85,B 0,C 180,E1 -12863.441,E2 -12863.441} C_VEL
LIN {X 0,Y 369.289,Z 298.485,A -85,B 0,C 180,E1 -12867.819,E2 -12867.819} C_VEL
LIN {X 0,Y 369.189,Z 298.494,A -85,B 0,C 180,E1 -12871.091,E2 -12871.091} C_VEL
LIN {X 0,Y 369.29,Z 298.485,A -85,B 0,C 180,E1 -12872.181,E2 -12872.181} C_VEL
LIN {X 0,Y 369.149,Z 298.5,A -85,B 0,C 180,E1 -12876.559,E2 -12876.559} C_VEL
LIN {X 0,Y 369.051,Z 298.516,A -85,B 0,C 180,E1 -12879.869,E2 -12879.869} C_VEL
LIN {X 0,Y 369.025,Z 298.519,A -85,B 0,C 180,E1 -12883.773,E2 -12883.773} C_VEL
LIN {X 0,Y 368.99,Z 298.523,A -85,B 0,C 180,E1 -12887.769,E2 -12887.769} C_VEL
LIN {X 0,Y 368.918,Z 298.532,A -85,B 0,C 180,E1 -12891.22,E2 -12891.22} C_VEL
LIN {X 0,Y 368.947,Z 298.526,A -85,B 0,C 180,E1 -12894.776,E2 -12894.776} C_VEL
LIN {X 0,Y 368.977,Z 298.522,A -85,B 0,C 180,E1 -12898.436,E2 -12898.436} C_VEL
LIN {X 0,Y 368.891,Z 298.533,A -85,B 0,C 180,E1 -12902.239,E2 -12902.239} C_VEL
LIN {X 0,Y 368.92,Z 298.532,A -85,B 0,C 180,E1 -12905.003,E2 -12905.003} C_VEL
LIN {X 0,Y 368.902,Z 298.533,A -85,B 0,C 180,E1 -12908.642,E2 -12908.642} C_VEL
LIN {X 0,Y 368.873,Z 298.534,A -85,B 0,C 180,E1 -12912.011,E2 -12912.011} C_VEL
LIN {X 0,Y 368.859,Z 298.536,A -85,B 0,C 180,E1 -12913.919,E2 -12913.919} C_VEL
LIN {X 0,Y 368.178,Z 298.624,A -85,B 0,C 180,E1 -12914.83,E2 -12914.83} C_VEL
LIN {X 0,Y 365.331,Z 298.978,A -85,B 0,C 180,E1 -12916.313,E2 -12916.313} C_VEL
LIN {X 0,Y 362.925,Z 299.28,A -85,B 0,C 180,E1 -12917.512,E2 -12917.512} C_VEL
LIN {X 0,Y 361.89,Z 299.408,A -85,B 0,C 180,E1 -12918.439,E2 -12918.439} C_VEL
LIN {X 0,Y 361.803,Z 299.417,A -85,B 0,C 180,E1 -12918.753,E2 -12918.753} C_VEL
LIN {X 0,Y 361.836,Z 299.411,A -85,B 0,C 180,E1 -12921.574,E2 -12921.574} C_VEL
LIN {X 0,Y 361.868,Z 299.411,A -85,B 0,C 180,E1 -12924.657,E2 -12924.657} C_VEL
LIN {X 0,Y 362.062,Z 299.471,A -85,B 0,C 180,E1 -12928.769,E2 -12928.769} C_VEL
LIN {X 0,Y 362.141,Z 303.185,A -85,B 0,C 180,E1 -12930.978,E2 -12930.978} C_VEL
LIN {X 0,Y 361.707,Z 309.622,A -85,B 0,C 180,E1 -12934.695,E2 -12934.695} C_VEL
LIN {X 0,Y 361.441,Z 316.023,A -85,B 0,C 180,E1 -12938.321,E2 -12938.321} C_VEL
LIN {X 0,Y 361.179,Z 322.392,A -85,B 0,C 180,E1 -12941.862,E2 -12941.862} C_VEL
LIN {X 0,Y 360.975,Z 328.763,A -85,B 0,C 180,E1 -12945.34,E2 -12945.34} C_VEL
LIN {X 0,Y 360.891,Z 334.846,A -85,B 0,C 180,E1 -12948.594,E2 -12948.594} C_VEL
LIN {X 0,Y 362.227,Z 346.239,A -85,B 0,C 180,E1 -12949.309,E2 -12949.309} C_VEL
LIN {X 0,Y 362.798,Z 352.676,A -85,B 0,C 180,E1 -12949.82,E2 -12949.82} C_VEL
LIN {X 0,Y 362.352,Z 362.801,A -85,B 0,C 180,E1 -12950.794,E2 -12950.794} C_VEL
LIN {X 0,Y 361.976,Z 372.252,A -85,B 0,C 180,E1 -12951.973,E2 -12951.973} C_VEL
LIN {X 0,Y 361.688,Z 380.499,A -85,B 0,C 180,E1 -12953.306,E2 -12953.306} C_VEL
LIN {X 0,Y 361.439,Z 387.179,A -85,B 0,C 180,E1 -12954.702,E2 -12954.702} C_VEL
LIN {X 0,Y 361.203,Z 392.325,A -85,B 0,C 180,E1 -12956.097,E2 -12956.097} C_VEL
LIN {X 0,Y 360.894,Z 396.802,A -85,B 0,C 180,E1 -12957.769,E2 -12957.769} C_VEL
LIN {X 0,Y 360.884,Z 398.865,A -85,B 0,C 180,E1 -12958.886,E2 -12958.886} C_VEL
LIN {X 0,Y 360.865,Z 400.252,A -85,B 0,C 180,E1 -12960.001,E2 -12960.001} C_VEL
LIN {X 0,Y 360.932,Z 400.971,A -85,B 0,C 180,E1 -12961.117,E2 -12961.117} C_VEL
LIN {X 0,Y 361.086,Z 401.024,A -85,B 0,C 180,E1 -12962.232,E2 -12962.232} C_VEL
LIN {X 0,Y 361.36,Z 400.424,A -85,B 0,C 180,E1 -12963.346,E2 -12963.346} C_VEL
LIN {X 0,Y 361.788,Z 399.171,A -85,B 0,C 180,E1 -12964.458,E2 -12964.458} C_VEL
LIN {X 0,Y 362.567,Z 396.025,A -85,B 0,C 180,E1 -12966.121,E2 -12966.121} C_VEL
LIN {X 0,Y 363.433,Z 391.247,A -85,B 0,C 180,E1 -12967.781,E2 -12967.781} C_VEL
LIN {X 0,Y 364.313,Z 385.807,A -85,B 0,C 180,E1 -12969.159,E2 -12969.159} C_VEL
LIN {X 0,Y 365.382,Z 378.812,A -85,B 0,C 180,E1 -12970.53,E2 -12970.53} C_VEL
LIN {X 0,Y 366.646,Z 370.015,A -85,B 0,C 180,E1 -12971.865,E2 -12971.865} C_VEL
LIN {X 0,Y 367.501,Z 360.933,A -85,B 0,C 180,E1 -12972.958,E2 -12972.958} C_VEL
LIN {X 0,Y 365.714,Z 350.809,A -85,B 0,C 180,E1 -12974.13,E2 -12974.13} C_VEL
LIN {X 0,Y 362.528,Z 339.927,A -85,B 0,C 180,E1 -12975.307,E2 -12975.307} C_VEL
LIN {X 0,Y 363.068,Z 334.156,A -85,B 0,C 180,E1 -12979.214,E2 -12979.214} C_VEL
LIN {X 0,Y 363.73,Z 329.309,A -85,B 0,C 180,E1 -12982.734,E2 -12982.734} C_VEL
LIN {X 0,Y 364.491,Z 324.79,A -85,B 0,C 180,E1 -12986.327,E2 -12986.327} C_VEL
LIN {X 0,Y 365.14,Z 322.034,A -85,B 0,C 180,E1 -12988.764,E2 -12988.764} C_VEL
LIN {X 0,Y 365.529,Z 319.534,A -85,B 0,C 180,E1 -12991.275,E2 -12991.275} C_VEL
LIN {X 0,Y 365.669,Z 317.232,A -85,B 0,C 180,E1 -12994.265,E2 -12994.265} C_VEL
LIN {X 0,Y 365.564,Z 315.968,A -85,B 0,C 180,E1 -12996.584,E2 -12996.584} C_VEL
LIN {X 0,Y 365.52,Z 314.992,A -85,B 0,C 180,E1 -12999.727,E2 -12999.727} C_VEL
LIN {X 0,Y 365.587,Z 314.845,A -85,B 0,C 180,E1 -13002.288,E2 -13002.288} C_VEL
LIN {X 0,Y 365.861,Z 315.63,A -85,B 0,C 180,E1 -13005.297,E2 -13005.297} C_VEL
LIN {X 0,Y 366.418,Z 317.499,A -85,B 0,C 180,E1 -13008.422,E2 -13008.422} C_VEL
LIN {X 0,Y 367.216,Z 320.719,A -85,B 0,C 180,E1 -13011.693,E2 -13011.693} C_VEL
LIN {X 0,Y 368.065,Z 324.445,A -85,B 0,C 180,E1 -13014.382,E2 -13014.382} C_VEL
LIN {X 0,Y 369.011,Z 328.719,A -85,B 0,C 180,E1 -13016.931,E2 -13016.931} C_VEL
LIN {X 0,Y 369.587,Z 333.111,A -85,B 0,C 180,E1 -13019.107,E2 -13019.107} C_VEL
LIN {X 0,Y 368.457,Z 337.719,A -85,B 0,C 180,E1 -13020.897,E2 -13020.897} C_VEL
LIN {X 0,Y 365.989,Z 347.963,A -85,B 0,C 180,E1 -13024.495,E2 -13024.495} C_VEL
LIN {X 0,Y 364.212,Z 358.408,A -85,B 0,C 180,E1 -13027.857,E2 -13027.857} C_VEL
LIN {X 0,Y 363.549,Z 363.507,A -85,B 0,C 180,E1 -13029.415,E2 -13029.415} C_VEL
LIN {X 0,Y 366.144,Z 377.145,A -85,B 0,C 180,E1 -13030.235,E2 -13030.235} C_VEL
LIN {X 0,Y 367.062,Z 388.466,A -85,B 0,C 180,E1 -13031.005,E2 -13031.005} C_VEL
LIN {X 0,Y 366.955,Z 399.384,A -85,B 0,C 180,E1 -13031.867,E2 -13031.867} C_VEL
LIN {X 0,Y 365.638,Z 411.115,A -85,B 0,C 180,E1 -13032.955,E2 -13032.955} C_VEL
LIN {X 0,Y 364.294,Z 421.622,A -85,B 0,C 180,E1 -13034.187,E2 -13034.187} C_VEL
LIN {X 0,Y 363.1,Z 432.039,A -85,B 0,C 180,E1 -13035.713,E2 -13035.713} C_VEL
LIN {X 0,Y 362.04,Z 441.121,A -85,B 0,C 180,E1 -13037.386,E2 -13037.386} C_VEL
LIN {X 0,Y 361.232,Z 448.496,A -85,B 0,C 180,E1 -13039.065,E2 -13039.065} C_VEL
LIN {X 0,Y 360.893,Z 453.495,A -85,B 0,C 180,E1 -13040.472,E2 -13040.472} C_VEL
LIN {X 0,Y 360.684,Z 458.384,A -85,B 0,C 180,E1 -13042.161,E2 -13042.161} C_VEL
LIN {X 0,Y 360.606,Z 461.842,A -85,B 0,C 180,E1 -13043.706,E2 -13043.706} C_VEL
LIN {X 0,Y 360.601,Z 464.805,A -85,B 0,C 180,E1 -13045.529,E2 -13045.529} C_VEL
LIN {X 0,Y 360.751,Z 466.024,A -85,B 0,C 180,E1 -13046.649,E2 -13046.649} C_VEL
LIN {X 0,Y 360.836,Z 466.821,A -85,B 0,C 180,E1 -13047.768,E2 -13047.768} C_VEL
LIN {X 0,Y 360.836,Z 467.194,A -85,B 0,C 180,E1 -13048.884,E2 -13048.884} C_VEL
LIN {X 0,Y 360.804,Z 467.084,A -85,B 0,C 180,E1 -13050,E2 -13050} C_VEL
LIN {X 0,Y 360.838,Z 466.556,A -85,B 0,C 180,E1 -13051.116,E2 -13051.116} C_VEL
LIN {X 0,Y 360.944,Z 465.614,A -85,B 0,C 180,E1 -13052.232,E2 -13052.232} C_VEL
LIN {X 0,Y 360.864,Z 464.145,A -85,B 0,C 180,E1 -13053.35,E2 -13053.35} C_VEL
LIN {X 0,Y 360.73,Z 461.054,A -85,B 0,C 180,E1 -13055.03,E2 -13055.03} C_VEL
LIN {X 0,Y 360.816,Z 456.81,A -85,B 0,C 180,E1 -13056.711,E2 -13056.711} C_VEL
LIN {X 0,Y 360.851,Z 451.242,A -85,B 0,C 180,E1 -13058.399,E2 -13058.399} C_VEL
LIN {X 0,Y 361.05,Z 444.117,A -85,B 0,C 180,E1 -13060.09,E2 -13060.09} C_VEL
LIN {X 0,Y 361.546,Z 435.148,A -85,B 0,C 180,E1 -13061.777,E2 -13061.777} C_VEL
LIN {X 0,Y 362.181,Z 425.772,A -85,B 0,C 180,E1 -13063.18,E2 -13063.18} C_VEL
LIN {X 0,Y 362.644,Z 416.56,A -85,B 0,C 180,E1 -13064.301,E2 -13064.301} C_VEL
LIN {X 0,Y 363.333,Z 405.098,A -85,B 0,C 180,E1 -13065.425,E2 -13065.425} C_VEL
LIN {X 0,Y 363.907,Z 394.023,A -85,B 0,C 180,E1 -13066.262,E2 -13066.262} C_VEL
LIN {X 0,Y 362.966,Z 381.199,A -85,B 0,C 180,E1 -13067.016,E2 -13067.016} C_VEL
LIN {X 0,Y 362.085,Z 368.741,A -85,B 0,C 180,E1 -13067.522,E2 -13067.522} C_VEL
LIN {X 0,Y 361.916,Z 365.414,A -85,B 0,C 180,E1 -13067.663,E2 -13067.663} C_VEL
LIN {X 0,Y 363.262,Z 349.888,A -85,B 0,C 180,E1 -13072.105,E2 -13072.105} C_VEL
LIN {X 0,Y 364.982,Z 335.414,A -85,B 0,C 180,E1 -13076.288,E2 -13076.288} C_VEL
LIN {X 0,Y 366.507,Z 324.156,A -85,B 0,C 180,E1 -13079.589,E2 -13079.589} C_VEL
LIN {X 0,Y 366.258,Z 320.491,A -85,B 0,C 180,E1 -13080.721,E2 -13080.721} C_VEL
LIN {X 0,Y 364.124,Z 310.337,A -85,B 0,C 180,E1 -13084.037,E2 -13084.037} C_VEL
LIN {X 0,Y 361.901,Z 299.407,A -85,B 0,C 180,E1 -13087.79,E2 -13087.79} C_VEL
LIN {X 0,Y 361.833,Z 299.412,A -85,B 0,C 180,E1 -13091.33,E2 -13091.33} C_VEL
LIN {X 0,Y 361.823,Z 299.415,A -85,B 0,C 180,E1 -13094.368,E2 -13094.368} C_VEL
LIN {X 0,Y 361.841,Z 299.414,A -85,B 0,C 180,E1 -13097.567,E2 -13097.567} C_VEL
LIN {X 0,Y 361.875,Z 299.408,A -85,B 0,C 180,E1 -13100.973,E2 -13100.973} C_VEL
LIN {X 0,Y 361.894,Z 299.43,A -85,B 0,C 180,E1 -13103.85,E2 -13103.85} C_VEL
LIN {X 0,Y 363.024,Z 303.908,A -85,B 0,C 180,E1 -13106.353,E2 -13106.353} C_VEL
LIN {X 0,Y 364.135,Z 309.359,A -85,B 0,C 180,E1 -13109.237,E2 -13109.237} C_VEL
LIN {X 0,Y 364.335,Z 313.262,A -85,B 0,C 180,E1 -13111.166,E2 -13111.166} C_VEL
LIN {X 0,Y 363.833,Z 321.054,A -85,B 0,C 180,E1 -13114.85,E2 -13114.85} C_VEL
LIN {X 0,Y 363.55,Z 328.776,A -85,B 0,C 180,E1 -13118.45,E2 -13118.45} C_VEL
LIN {X 0,Y 363.179,Z 337.464,A -85,B 0,C 180,E1 -13122.544,E2 -13122.544} C_VEL
LIN {X 0,Y 362.952,Z 346.639,A -85,B 0,C 180,E1 -13126.883,E2 -13126.883} C_VEL
LIN {X 0,Y 365.543,Z 357.023,A -85,B 0,C 180,E1 -13127.789,E2 -13127.789} C_VEL
LIN {X 0,Y 365.899,Z 360.59,A -85,B 0,C 180,E1 -13128.111,E2 -13128.111} C_VEL
LIN {X 0,Y 365.299,Z 368.666,A -85,B 0,C 180,E1 -13128.906,E2 -13128.906} C_VEL
LIN {X 0,Y 364.417,Z 377.208,A -85,B 0,C 180,E1 -13130.003,E2 -13130.003} C_VEL
LIN {X 0,Y 363.791,Z 383.745,A -85,B 0,C 180,E1 -13131.108,E2 -13131.108} C_VEL
LIN {X 0,Y 363.269,Z 388.815,A -85,B 0,C 180,E1 -13132.215,E2 -13132.215} C_VEL
LIN {X 0,Y 362.701,Z 392.797,A -85,B 0,C 180,E1 -13133.322,E2 -13133.322} C_VEL
LIN {X 0,Y 362.234,Z 395.878,A -85,B 0,C 180,E1 -13134.432,E2 -13134.432} C_VEL
LIN {X 0,Y 361.766,Z 398.163,A -85,B 0,C 180,E1 -13135.542,E2 -13135.542} C_VEL
LIN {X 0,Y 361.325,Z 399.706,A -85,B 0,C 180,E1 -13136.653,E2 -13136.653} C_VEL
LIN {X 0,Y 361.055,Z 400.526,A -85,B 0,C 180,E1 -13137.767,E2 -13137.767} C_VEL
LIN {X 0,Y 360.909,Z 400.638,A -85,B 0,C 180,E1 -13138.883,E2 -13138.883} C_VEL
LIN {X 0,Y 360.851,Z 400.048,A -85,B 0,C 180,E1 -13139.999,E2 -13139.999} C_VEL
LIN {X 0,Y 360.877,Z 397.843,A -85,B 0,C 180,E1 -13141.673,E2 -13141.673} C_VEL
LIN {X 0,Y 360.954,Z 395.484,A -85,B 0,C 180,E1 -13142.789,E2 -13142.789} C_VEL
LIN {X 0,Y 361.179,Z 392.284,A -85,B 0,C 180,E1 -13143.904,E2 -13143.904} C_VEL
LIN {X 0,Y 361.374,Z 386.941,A -85,B 0,C 180,E1 -13145.299,E2 -13145.299} C_VEL
LIN {X 0,Y 361.569,Z 381.458,A -85,B 0,C 180,E1 -13146.416,E2 -13146.416} C_VEL
LIN {X 0,Y 361.677,Z 375.556,A -85,B 0,C 180,E1 -13147.366,E2 -13147.366} C_VEL
LIN {X 0,Y 361.874,Z 367.81,A -85,B 0,C 180,E1 -13148.374,E2 -13148.374} C_VEL
LIN {X 0,Y 362.1,Z 359.351,A -85,B 0,C 180,E1 -13149.213,E2 -13149.213} C_VEL
LIN {X 0,Y 362.283,Z 350.102,A -85,B 0,C 180,E1 -13149.912,E2 -13149.912} C_VEL
LIN {X 0,Y 361.332,Z 342.514,A -85,B 0,C 180,E1 -13150.363,E2 -13150.363} C_VEL
LIN {X 0,Y 361.442,Z 335.296,A -85,B 0,C 180,E1 -13153.537,E2 -13153.537} C_VEL
LIN {X 0,Y 361.469,Z 327.639,A -85,B 0,C 180,E1 -13156.955,E2 -13156.955} C_VEL
LIN {X 0,Y 361.578,Z 319.816,A -85,B 0,C 180,E1 -13160.477,E2 -13160.477} C_VEL
LIN {X 0,Y 361.738,Z 311.87,A -85,B 0,C 180,E1 -13164.077,E2 -13164.077} C_VEL
LIN {X 0,Y 361.848,Z 303.674,A -85,B 0,C 180,E1 -13167.782,E2 -13167.782} C_VEL
LIN {X 0,Y 361.993,Z 299.393,A -85,B 0,C 180,E1 -13169.752,E2 -13169.752} C_VEL
LIN {X 0,Y 361.848,Z 299.408,A -85,B 0,C 180,E1 -13174.279,E2 -13174.279} C_VEL
LIN {X 0,Y 361.854,Z 299.413,A -85,B 0,C 180,E1 -13177.22,E2 -13177.22} C_VEL
LIN {X 0,Y 361.806,Z 299.417,A -85,B 0,C 180,E1 -13180.75,E2 -13180.75} C_VEL
LIN {X 0,Y 361.809,Z 299.415,A -85,B 0,C 180,E1 -13184.367,E2 -13184.367} C_VEL
LIN {X 0,Y 361.828,Z 299.413,A -85,B 0,C 180,E1 -13187.567,E2 -13187.567} C_VEL
LIN {X 0,Y 361.863,Z 299.411,A -85,B 0,C 180,E1 -13190.972,E2 -13190.972} C_VEL
LIN {X 0,Y 361.866,Z 299.412,A -85,B 0,C 180,E1 -13194.654,E2 -13194.654} C_VEL
LIN {X 0,Y 361.829,Z 299.415,A -85,B 0,C 180,E1 -13198.37,E2 -13198.37} C_VEL
LIN {X 0,Y 361.893,Z 299.407,A -85,B 0,C 180,E1 -13200.954,E2 -13200.954} C_VEL
LIN {X 0,Y 361.944,Z 299.398,A -85,B 0,C 180,E1 -13203.474,E2 -13203.474} C_VEL
LIN {X 0,Y 361.879,Z 299.407,A -85,B 0,C 180,E1 -13207.144,E2 -13207.144} C_VEL
LIN {X 0,Y 361.91,Z 299.405,A -85,B 0,C 180,E1 -13210.723,E2 -13210.723} C_VEL
LIN {X 0,Y 361.934,Z 299.402,A -85,B 0,C 180,E1 -13214.226,E2 -13214.226} C_VEL
LIN {X 0,Y 361.987,Z 299.396,A -85,B 0,C 180,E1 -13216.527,E2 -13216.527} C_VEL
LIN {X 0,Y 361.988,Z 299.395,A -85,B 0,C 180,E1 -13219.937,E2 -13219.937} C_VEL
LIN {X 0,Y 362.112,Z 299.376,A -85,B 0,C 180,E1 -13223.313,E2 -13223.313} C_VEL
LIN {X 0,Y 362.253,Z 299.361,A -85,B 0,C 180,E1 -13227.776,E2 -13227.776} C_VEL
LIN {X 0,Y 362.16,Z 299.37,A -85,B 0,C 180,E1 -13231.112,E2 -13231.112} C_VEL
LIN {X 0,Y 362.253,Z 299.361,A -85,B 0,C 180,E1 -13232.224,E2 -13232.224} C_VEL
LIN {X 0,Y 362.112,Z 299.376,A -85,B 0,C 180,E1 -13236.687,E2 -13236.687} C_VEL
LIN {X 0,Y 361.988,Z 299.395,A -85,B 0,C 180,E1 -13240.063,E2 -13240.063} C_VEL
LIN {X 0,Y 361.986,Z 299.395,A -85,B 0,C 180,E1 -13243.899,E2 -13243.899} C_VEL
LIN {X 0,Y 361.956,Z 299.399,A -85,B 0,C 180,E1 -13247.939,E2 -13247.939} C_VEL
LIN {X 0,Y 361.881,Z 299.409,A -85,B 0,C 180,E1 -13251.654,E2 -13251.654} C_VEL
LIN {X 0,Y 361.918,Z 299.405,A -85,B 0,C 180,E1 -13255.291,E2 -13255.291} C_VEL
LIN {X 0,Y 361.912,Z 299.404,A -85,B 0,C 180,E1 -13257.779,E2 -13257.779} C_VEL
LIN {X 0,Y 361.837,Z 299.415,A -85,B 0,C 180,E1 -13261.286,E2 -13261.286} C_VEL
LIN {X 0,Y 361.845,Z 299.41,A -85,B 0,C 180,E1 -13264.282,E2 -13264.282} C_VEL
LIN {X 0,Y 361.863,Z 299.412,A -85,B 0,C 180,E1 -13267.226,E2 -13267.226} C_VEL
LIN {X 0,Y 361.828,Z 299.415,A -85,B 0,C 180,E1 -13270.757,E2 -13270.757} C_VEL
LIN {X 0,Y 361.809,Z 299.415,A -85,B 0,C 180,E1 -13274.37,E2 -13274.37} C_VEL
LIN {X 0,Y 361.823,Z 299.413,A -85,B 0,C 180,E1 -13277.571,E2 -13277.571} C_VEL
LIN {X 0,Y 361.803,Z 299.417,A -85,B 0,C 180,E1 -13278.753,E2 -13278.753} C_VEL
LIN {X 0,Y 361.131,Z 299.5,A -85,B 0,C 180,E1 -13279.682,E2 -13279.682} C_VEL
LIN {X 0,Y 358.286,Z 299.855,A -85,B 0,C 180,E1 -13281.193,E2 -13281.193} C_VEL
LIN {X 0,Y 355.887,Z 300.153,A -85,B 0,C 180,E1 -13282.416,E2 -13282.416} C_VEL
LIN {X 0,Y 354.867,Z 300.28,A -85,B 0,C 180,E1 -13283.361,E2 -13283.361} C_VEL
LIN {X 0,Y 354.789,Z 300.288,A -85,B 0,C 180,E1 -13283.681,E2 -13283.681} C_VEL
LIN {X 0,Y 354.853,Z 300.28,A -85,B 0,C 180,E1 -13287.676,E2 -13287.676} C_VEL
LIN {X 0,Y 355.003,Z 300.328,A -85,B 0,C 180,E1 -13288.698,E2 -13288.698} C_VEL
LIN {X 0,Y 355.084,Z 303.411,A -85,B 0,C 180,E1 -13290.56,E2 -13290.56} C_VEL
LIN {X 0,Y 354.717,Z 309.541,A -85,B 0,C 180,E1 -13294.16,E2 -13294.16} C_VEL
LIN {X 0,Y 354.41,Z 316.004,A -85,B 0,C 180,E1 -13297.868,E2 -13297.868} C_VEL
LIN {X 0,Y 354.202,Z 321.346,A -85,B 0,C 180,E1 -13300.891,E2 -13300.891} C_VEL
LIN {X 0,Y 353.968,Z 327.765,A -85,B 0,C 180,E1 -13304.454,E2 -13304.454} C_VEL
LIN {X 0,Y 353.833,Z 334.211,A -85,B 0,C 180,E1 -13307.964,E2 -13307.964} C_VEL
LIN {X 0,Y 353.84,Z 335.328,A -85,B 0,C 180,E1 -13308.473,E2 -13308.473} C_VEL
LIN {X 0,Y 355.089,Z 346.234,A -85,B 0,C 180,E1 -13309.164,E2 -13309.164} C_VEL
LIN {X 0,Y 355.745,Z 351.919,A -85,B 0,C 180,E1 -13309.616,E2 -13309.616} C_VEL
LIN {X 0,Y 355.303,Z 362.274,A -85,B 0,C 180,E1 -13310.61,E2 -13310.61} C_VEL
LIN {X 0,Y 354.941,Z 371.837,A -85,B 0,C 180,E1 -13311.803,E2 -13311.803} C_VEL
LIN {X 0,Y 354.676,Z 379.119,A -85,B 0,C 180,E1 -13312.95,E2 -13312.95} C_VEL
LIN {X 0,Y 354.39,Z 385.999,A -85,B 0,C 180,E1 -13314.311,E2 -13314.311} C_VEL
LIN {X 0,Y 354.141,Z 390.586,A -85,B 0,C 180,E1 -13315.449,E2 -13315.449} C_VEL
LIN {X 0,Y 353.998,Z 394.29,A -85,B 0,C 180,E1 -13316.587,E2 -13316.587} C_VEL
LIN {X 0,Y 353.798,Z 398.369,A -85,B 0,C 180,E1 -13318.294,E2 -13318.294} C_VEL
LIN {X 0,Y 353.814,Z 400.841,A -85,B 0,C 180,E1 -13320.001,E2 -13320.001} C_VEL
LIN {X 0,Y 353.882,Z 401.656,A -85,B 0,C 180,E1 -13321.139,E2 -13321.139} C_VEL
LIN {X 0,Y 354.043,Z 401.821,A -85,B 0,C 180,E1 -13322.277,E2 -13322.277} C_VEL
LIN {X 0,Y 354.332,Z 401.339,A -85,B 0,C 180,E1 -13323.413,E2 -13323.413} C_VEL
LIN {X 0,Y 354.784,Z 400.199,A -85,B 0,C 180,E1 -13324.546,E2 -13324.546} C_VEL
LIN {X 0,Y 355.604,Z 397.225,A -85,B 0,C 180,E1 -13326.242,E2 -13326.242} C_VEL
LIN {X 0,Y 356.534,Z 392.649,A -85,B 0,C 180,E1 -13327.933,E2 -13327.933} C_VEL
LIN {X 0,Y 357.492,Z 387.486,A -85,B 0,C 180,E1 -13329.335,E2 -13329.335} C_VEL
LIN {X 0,Y 358.619,Z 380.793,A -85,B 0,C 180,E1 -13330.731,E2 -13330.731} C_VEL
LIN {X 0,Y 359.958,Z 372.134,A -85,B 0,C 180,E1 -13332.117,E2 -13332.117} C_VEL
LIN {X 0,Y 361.017,Z 363.161,A -85,B 0,C 180,E1 -13333.254,E2 -13333.254} C_VEL
LIN {X 0,Y 359.674,Z 354.24,A -85,B 0,C 180,E1 -13334.372,E2 -13334.372} C_VEL
LIN {X 0,Y 356.657,Z 343.647,A -85,B 0,C 180,E1 -13335.591,E2 -13335.591} C_VEL
LIN {X 0,Y 355.643,Z 340.539,A -85,B 0,C 180,E1 -13335.93,E2 -13335.93} C_VEL
LIN {X 0,Y 356.223,Z 335.307,A -85,B 0,C 180,E1 -13339.598,E2 -13339.598} C_VEL
LIN {X 0,Y 356.934,Z 330.528,A -85,B 0,C 180,E1 -13343.192,E2 -13343.192} C_VEL
LIN {X 0,Y 357.78,Z 326.12,A -85,B 0,C 180,E1 -13346.86,E2 -13346.86} C_VEL
LIN {X 0,Y 358.434,Z 323.461,A -85,B 0,C 180,E1 -13349.354,E2 -13349.354} C_VEL
LIN {X 0,Y 358.831,Z 321.17,A -85,B 0,C 180,E1 -13351.927,E2 -13351.927} C_VEL
LIN {X 0,Y 358.933,Z 319.247,A -85,B 0,C 180,E1 -13354.677,E2 -13354.677} C_VEL
LIN {X 0,Y 358.82,Z 317.966,A -85,B 0,C 180,E1 -13357.387,E2 -13357.387} C_VEL
LIN {X 0,Y 358.858,Z 317.335,A -85,B 0,C 180,E1 -13360.263,E2 -13360.263} C_VEL
LIN {X 0,Y 359.053,Z 317.583,A -85,B 0,C 180,E1 -13363.595,E2 -13363.595} C_VEL
LIN {X 0,Y 359.497,Z 318.971,A -85,B 0,C 180,E1 -13366.824,E2 -13366.824} C_VEL
LIN {X 0,Y 360.148,Z 321.386,A -85,B 0,C 180,E1 -13369.911,E2 -13369.911} C_VEL
LIN {X 0,Y 360.95,Z 324.902,A -85,B 0,C 180,E1 -13372.97,E2 -13372.97} C_VEL
LIN {X 0,Y 361.867,Z 328.987,A -85,B 0,C 180,E1 -13375.721,E2 -13375.721} C_VEL
LIN {X 0,Y 362.76,Z 334.094,A -85,B 0,C 180,E1 -13378.48,E2 -13378.48} C_VEL
LIN {X 0,Y 362.743,Z 335.435,A -85,B 0,C 180,E1 -13379.117,E2 -13379.117} C_VEL
LIN {X 0,Y 361.023,Z 341.765,A -85,B 0,C 180,E1 -13381.581,E2 -13381.581} C_VEL
LIN {X 0,Y 358.671,Z 351.681,A -85,B 0,C 180,E1 -13385.084,E2 -13385.084} C_VEL
LIN {X 0,Y 357.116,Z 360.696,A -85,B 0,C 180,E1 -13388.042,E2 -13388.042} C_VEL
LIN {X 0,Y 356.765,Z 363.043,A -85,B 0,C 180,E1 -13388.778,E2 -13388.778} C_VEL
LIN {X 0,Y 359.473,Z 376.625,A -85,B 0,C 180,E1 -13389.662,E2 -13389.662} C_VEL
LIN {X 0,Y 360.485,Z 387.216,A -85,B 0,C 180,E1 -13390.421,E2 -13390.421} C_VEL
LIN {X 0,Y 360.419,Z 398.939,A -85,B 0,C 180,E1 -13391.379,E2 -13391.379} C_VEL
LIN {X 0,Y 359.104,Z 410.544,A -85,B 0,C 180,E1 -13392.488,E2 -13392.488} C_VEL
LIN {X 0,Y 357.63,Z 420.986,A -85,B 0,C 180,E1 -13393.738,E2 -13393.738} C_VEL
LIN {X 0,Y 356.415,Z 430.474,A -85,B 0,C 180,E1 -13395.147,E2 -13395.147} C_VEL
LIN {X 0,Y 355.404,Z 438.327,A -85,B 0,C 180,E1 -13396.564,E2 -13396.564} C_VEL
LIN {X 0,Y 354.514,Z 446.041,A -85,B 0,C 180,E1 -13398.276,E2 -13398.276} C_VEL
LIN {X 0,Y 353.974,Z 451.329,A -85,B 0,C 180,E1 -13399.706,E2 -13399.706} C_VEL
LIN {X 0,Y 353.646,Z 456.492,A -85,B 0,C 180,E1 -13401.428,E2 -13401.428} C_VEL
LIN {X 0,Y 353.531,Z 460.502,A -85,B 0,C 180,E1 -13403.15,E2 -13403.15} C_VEL
LIN {X 0,Y 353.507,Z 462.592,A -85,B 0,C 180,E1 -13404.295,E2 -13404.295} C_VEL
LIN {X 0,Y 353.525,Z 464.216,A -85,B 0,C 180,E1 -13405.439,E2 -13405.439} C_VEL
LIN {X 0,Y 353.655,Z 465.392,A -85,B 0,C 180,E1 -13406.582,E2 -13406.582} C_VEL
LIN {X 0,Y 353.762,Z 466.153,A -85,B 0,C 180,E1 -13407.723,E2 -13407.723} C_VEL
LIN {X 0,Y 353.79,Z 466.461,A -85,B 0,C 180,E1 -13408.862,E2 -13408.862} C_VEL
LIN {X 0,Y 353.757,Z 466.306,A -85,B 0,C 180,E1 -13410,E2 -13410} C_VEL
LIN {X 0,Y 353.793,Z 465.74,A -85,B 0,C 180,E1 -13411.138,E2 -13411.138} C_VEL
LIN {X 0,Y 353.898,Z 464.72,A -85,B 0,C 180,E1 -13412.276,E2 -13412.276} C_VEL
LIN {X 0,Y 353.801,Z 463.22,A -85,B 0,C 180,E1 -13413.416,E2 -13413.416} C_VEL
LIN {X 0,Y 353.678,Z 460.035,A -85,B 0,C 180,E1 -13415.13,E2 -13415.13} C_VEL
LIN {X 0,Y 353.761,Z 455.675,A -85,B 0,C 180,E1 -13416.846,E2 -13416.846} C_VEL
LIN {X 0,Y 353.818,Z 449.964,A -85,B 0,C 180,E1 -13418.568,E2 -13418.568} C_VEL
LIN {X 0,Y 354.029,Z 442.659,A -85,B 0,C 180,E1 -13420.292,E2 -13420.292} C_VEL
LIN {X 0,Y 354.44,Z 435.155,A -85,B 0,C 180,E1 -13421.727,E2 -13421.727} C_VEL
LIN {X 0,Y 355.066,Z 425.97,A -85,B 0,C 180,E1 -13423.157,E2 -13423.157} C_VEL
LIN {X 0,Y 355.49,Z 417.227,A -85,B 0,C 180,E1 -13424.267,E2 -13424.267} C_VEL
LIN {X 0,Y 356.213,Z 405.682,A -85,B 0,C 180,E1 -13425.447,E2 -13425.447} C_VEL
LIN {X 0,Y 356.846,Z 395.054,A -85,B 0,C 180,E1 -13426.299,E2 -13426.299} C_VEL
LIN {X 0,Y 355.991,Z 382.482,A -85,B 0,C 180,E1 -13427.077,E2 -13427.077} C_VEL
LIN {X 0,Y 355.116,Z 370.091,A -85,B 0,C 180,E1 -13427.627,E2 -13427.627} C_VEL
LIN {X 0,Y 354.839,Z 365.315,A -85,B 0,C 180,E1 -13427.78,E2 -13427.78} C_VEL
LIN {X 0,Y 356.246,Z 349.856,A -85,B 0,C 180,E1 -13432.319,E2 -13432.319} C_VEL
LIN {X 0,Y 358.153,Z 334.666,A -85,B 0,C 180,E1 -13436.829,E2 -13436.829} C_VEL
LIN {X 0,Y 359.571,Z 324.466,A -85,B 0,C 180,E1 -13439.895,E2 -13439.895} C_VEL
LIN {X 0,Y 358.959,Z 320.228,A -85,B 0,C 180,E1 -13441.254,E2 -13441.254} C_VEL
LIN {X 0,Y 356.743,Z 309.567,A -85,B 0,C 180,E1 -13444.842,E2 -13444.842} C_VEL
LIN {X 0,Y 354.849,Z 300.286,A -85,B 0,C 180,E1 -13448.148,E2 -13448.148} C_VEL
LIN {X 0,Y 354.8,Z 300.292,A -85,B 0,C 180,E1 -13452.337,E2 -13452.337} C_VEL
LIN {X 0,Y 354.773,Z 300.293,A -85,B 0,C 180,E1 -13456.103,E2 -13456.103} C_VEL
LIN {X 0,Y 354.794,Z 300.291,A -85,B 0,C 180,E1 -13459.178,E2 -13459.178} C_VEL
LIN {X 0,Y 354.859,Z 300.432,A -85,B 0,C 180,E1 -13462.623,E2 -13462.623} C_VEL
LIN {X 0,Y 356.303,Z 305.942,A -85,B 0,C 180,E1 -13465.939,E2 -13465.939} C_VEL
LIN {X 0,Y 357.517,Z 311.979,A -85,B 0,C 180,E1 -13469.261,E2 -13469.261} C_VEL
LIN {X 0,Y 357.604,Z 315.821,A -85,B 0,C 180,E1 -13471.215,E2 -13471.215} C_VEL
LIN {X 0,Y 357.099,Z 323.446,A -85,B 0,C 180,E1 -13474.867,E2 -13474.867} C_VEL
LIN {X 0,Y 356.693,Z 331.239,A -85,B 0,C 180,E1 -13478.621,E2 -13478.621} C_VEL
LIN {X 0,Y 356.342,Z 338.689,A -85,B 0,C 180,E1 -13482.198,E2 -13482.198} C_VEL
LIN {X 0,Y 356.09,Z 347.4,A -85,B 0,C 180,E1 -13486.371,E2 -13486.371} C_VEL
LIN {X 0,Y 356.164,Z 347.883,A -85,B 0,C 180,E1 -13486.465,E2 -13486.465} C_VEL
LIN {X 0,Y 358.638,Z 356.909,A -85,B 0,C 180,E1 -13487.263,E2 -13487.263} C_VEL
LIN {X 0,Y 359.329,Z 361.604,A -85,B 0,C 180,E1 -13487.718,E2 -13487.718} C_VEL
LIN {X 0,Y 358.642,Z 370.04,A -85,B 0,C 180,E1 -13488.582,E2 -13488.582} C_VEL
LIN {X 0,Y 357.826,Z 377.366,A -85,B 0,C 180,E1 -13489.543,E2 -13489.543} C_VEL
LIN {X 0,Y 357.089,Z 383.89,A -85,B 0,C 180,E1 -13490.654,E2 -13490.654} C_VEL
LIN {X 0,Y 356.372,Z 390.219,A -85,B 0,C 180,E1 -13492.064,E2 -13492.064} C_VEL
LIN {X 0,Y 355.768,Z 394.087,A -85,B 0,C 180,E1 -13493.192,E2 -13493.192} C_VEL
LIN {X 0,Y 355.268,Z 397.061,A -85,B 0,C 180,E1 -13494.322,E2 -13494.322} C_VEL
LIN {X 0,Y 354.767,Z 399.231,A -85,B 0,C 180,E1 -13495.454,E2 -13495.454} C_VEL
LIN {X 0,Y 354.301,Z 400.646,A -85,B 0,C 180,E1 -13496.587,E2 -13496.587} C_VEL
LIN {X 0,Y 354.014,Z 401.335,A -85,B 0,C 180,E1 -13497.723,E2 -13497.723} C_VEL
LIN {X 0,Y 353.861,Z 401.325,A -85,B 0,C 180,E1 -13498.861,E2 -13498.861} C_VEL
LIN {X 0,Y 353.8,Z 400.624,A -85,B 0,C 180,E1 -13499.999,E2 -13499.999} C_VEL
LIN {X 0,Y 353.81,Z 398.311,A -85,B 0,C 180,E1 -13501.706,E2 -13501.706} C_VEL
LIN {X 0,Y 353.886,Z 395.816,A -85,B 0,C 180,E1 -13502.844,E2 -13502.844} C_VEL
LIN {X 0,Y 354.116,Z 392.457,A -85,B 0,C 180,E1 -13503.982,E2 -13503.982} C_VEL
LIN {X 0,Y 354.298,Z 386.975,A -85,B 0,C 180,E1 -13505.405,E2 -13505.405} C_VEL
LIN {X 0,Y 354.499,Z 381.233,A -85,B 0,C 180,E1 -13506.544,E2 -13506.544} C_VEL
LIN {X 0,Y 354.621,Z 375.144,A -85,B 0,C 180,E1 -13507.513,E2 -13507.513} C_VEL
LIN {X 0,Y 354.811,Z 367.067,A -85,B 0,C 180,E1 -13508.542,E2 -13508.542} C_VEL
LIN {X 0,Y 355.089,Z 358.208,A -85,B 0,C 180,E1 -13509.396,E2 -13509.396} C_VEL
LIN {X 0,Y 355.191,Z 350.515,A -85,B 0,C 180,E1 -13509.968,E2 -13509.968} C_VEL
LIN {X 0,Y 354.272,Z 343.101,A -85,B 0,C 180,E1 -13510.428,E2 -13510.428} C_VEL
LIN {X 0,Y 354.375,Z 335.548,A -85,B 0,C 180,E1 -13513.766,E2 -13513.766} C_VEL
LIN {X 0,Y 354.405,Z 327.66,A -85,B 0,C 180,E1 -13517.303,E2 -13517.303} C_VEL
LIN {X 0,Y 354.541,Z 319.71,A -85,B 0,C 180,E1 -13520.903,E2 -13520.903} C_VEL
LIN {X 0,Y 354.695,Z 311.665,A -85,B 0,C 180,E1 -13524.587,E2 -13524.587} C_VEL
LIN {X 0,Y 354.804,Z 304.736,A -85,B 0,C 180,E1 -13527.74,E2 -13527.74} C_VEL
LIN {X 0,Y 354.922,Z 300.273,A -85,B 0,C 180,E1 -13529.834,E2 -13529.834} C_VEL
LIN {X 0,Y 354.801,Z 300.288,A -85,B 0,C 180,E1 -13533.7,E2 -13533.7} C_VEL
LIN {X 0,Y 354.789,Z 300.288,A -85,B 0,C 180,E1 -13536.458,E2 -13536.458} C_VEL
LIN {X 0,Y 354.761,Z 300.295,A -85,B 0,C 180,E1 -13539.411,E2 -13539.411} C_VEL
LIN {X 0,Y 354.778,Z 300.294,A -85,B 0,C 180,E1 -13542.865,E2 -13542.865} C_VEL
LIN {X 0,Y 354.759,Z 300.292,A -85,B 0,C 180,E1 -13546.102,E2 -13546.102} C_VEL
LIN {X 0,Y 354.781,Z 300.293,A -85,B 0,C 180,E1 -13549.178,E2 -13549.178} C_VEL
LIN {X 0,Y 354.804,Z 300.289,A -85,B 0,C 180,E1 -13552.4,E2 -13552.4} C_VEL
LIN {X 0,Y 354.803,Z 300.291,A -85,B 0,C 180,E1 -13554.94,E2 -13554.94} C_VEL
LIN {X 0,Y 354.784,Z 300.292,A -85,B 0,C 180,E1 -13558.404,E2 -13558.404} C_VEL
LIN {X 0,Y 354.844,Z 300.282,A -85,B 0,C 180,E1 -13561.618,E2 -13561.618} C_VEL
LIN {X 0,Y 354.889,Z 300.279,A -85,B 0,C 180,E1 -13564.172,E2 -13564.172} C_VEL
LIN {X 0,Y 354.824,Z 300.285,A -85,B 0,C 180,E1 -13567.893,E2 -13567.893} C_VEL
LIN {X 0,Y 354.912,Z 300.275,A -85,B 0,C 180,E1 -13571.891,E2 -13571.891} C_VEL
LIN {X 0,Y 354.931,Z 300.274,A -85,B 0,C 180,E1 -13575.981,E2 -13575.981} C_VEL
LIN {X 0,Y 354.944,Z 300.271,A -85,B 0,C 180,E1 -13579.735,E2 -13579.735} C_VEL
LIN {X 0,Y 355.077,Z 300.252,A -85,B 0,C 180,E1 -13583.18,E2 -13583.18} C_VEL
LIN {X 0,Y 355.215,Z 300.238,A -85,B 0,C 180,E1 -13587.732,E2 -13587.732} C_VEL
LIN {X 0,Y 355.132,Z 300.245,A -85,B 0,C 180,E1 -13591.134,E2 -13591.134} C_VEL
LIN {X 0,Y 355.215,Z 300.238,A -85,B 0,C 180,E1 -13592.268,E2 -13592.268} C_VEL
LIN {X 0,Y 355.077,Z 300.252,A -85,B 0,C 180,E1 -13596.82,E2 -13596.82} C_VEL
LIN {X 0,Y 354.944,Z 300.271,A -85,B 0,C 180,E1 -13600.265,E2 -13600.265} C_VEL
LIN {X 0,Y 354.931,Z 300.274,A -85,B 0,C 180,E1 -13604.019,E2 -13604.019} C_VEL
LIN {X 0,Y 354.912,Z 300.275,A -85,B 0,C 180,E1 -13608.109,E2 -13608.109} C_VEL
LIN {X 0,Y 354.824,Z 300.285,A -85,B 0,C 180,E1 -13612.107,E2 -13612.107} C_VEL
LIN {X 0,Y 354.889,Z 300.279,A -85,B 0,C 180,E1 -13615.828,E2 -13615.828} C_VEL
LIN {X 0,Y 354.845,Z 300.285,A -85,B 0,C 180,E1 -13619.68,E2 -13619.68} C_VEL
LIN {X 0,Y 354.797,Z 300.29,A -85,B 0,C 180,E1 -13623.703,E2 -13623.703} C_VEL
LIN {X 0,Y 354.792,Z 300.289,A -85,B 0,C 180,E1 -13626.46,E2 -13626.46} C_VEL
LIN {X 0,Y 354.816,Z 300.288,A -85,B 0,C 180,E1 -13629.425,E2 -13629.425} C_VEL
LIN {X 0,Y 354.78,Z 300.293,A -85,B 0,C 180,E1 -13632.869,E2 -13632.869} C_VEL
LIN {X 0,Y 354.759,Z 300.292,A -85,B 0,C 180,E1 -13636.105,E2 -13636.105} C_VEL
LIN {X 0,Y 354.759,Z 300.295,A -85,B 0,C 180,E1 -13639.178,E2 -13639.178} C_VEL
LIN {X 0,Y 354.794,Z 300.289,A -85,B 0,C 180,E1 -13642.406,E2 -13642.406} C_VEL
LIN {X 0,Y 354.789,Z 300.288,A -85,B 0,C 180,E1 -13643.681,E2 -13643.681} C_VEL
LIN {X 0,Y 354.127,Z 300.446,A -85,B 0,C 180,E1 -13644.636,E2 -13644.636} C_VEL
LIN {X 0,Y 351.276,Z 300.727,A -85,B 0,C 180,E1 -13646.191,E2 -13646.191} C_VEL
LIN {X 0,Y 348.937,Z 301.017,A -85,B 0,C 180,E1 -13647.439,E2 -13647.439} C_VEL
LIN {X 0,Y 347.983,Z 301.169,A -85,B 0,C 180,E1 -13648.552,E2 -13648.552} C_VEL
LIN {X 0,Y 347.99,Z 301.317,A -85,B 0,C 180,E1 -13648.708,E2 -13648.708} C_VEL
LIN {X 0,Y 348.076,Z 303.836,A -85,B 0,C 180,E1 -13650.252,E2 -13650.252} C_VEL
LIN {X 0,Y 347.702,Z 309.461,A -85,B 0,C 180,E1 -13653.599,E2 -13653.599} C_VEL
LIN {X 0,Y 347.406,Z 315.954,A -85,B 0,C 180,E1 -13657.397,E2 -13657.397} C_VEL
LIN {X 0,Y 347.111,Z 322.415,A -85,B 0,C 180,E1 -13661.1,E2 -13661.1} C_VEL
LIN {X 0,Y 346.876,Z 328.881,A -85,B 0,C 180,E1 -13664.73,E2 -13664.73} C_VEL
LIN {X 0,Y 346.764,Z 335.544,A -85,B 0,C 180,E1 -13668.345,E2 -13668.345} C_VEL
LIN {X 0,Y 347.886,Z 345.963,A -85,B 0,C 180,E1 -13669.011,E2 -13669.011} C_VEL
LIN {X 0,Y 348.675,Z 352.613,A -85,B 0,C 180,E1 -13669.55,E2 -13669.55} C_VEL
LIN {X 0,Y 348.222,Z 362.918,A -85,B 0,C 180,E1 -13670.563,E2 -13670.563} C_VEL
LIN {X 0,Y 347.878,Z 372.087,A -85,B 0,C 180,E1 -13671.726,E2 -13671.726} C_VEL
LIN {X 0,Y 347.576,Z 380.214,A -85,B 0,C 180,E1 -13673.033,E2 -13673.033} C_VEL
LIN {X 0,Y 347.283,Z 387.285,A -85,B 0,C 180,E1 -13674.485,E2 -13674.485} C_VEL
LIN {X 0,Y 347.074,Z 392.75,A -85,B 0,C 180,E1 -13675.937,E2 -13675.937} C_VEL
LIN {X 0,Y 346.762,Z 397.546,A -85,B 0,C 180,E1 -13677.678,E2 -13677.678} C_VEL
LIN {X 0,Y 346.726,Z 399.815,A -85,B 0,C 180,E1 -13678.84,E2 -13678.84} C_VEL
LIN {X 0,Y 346.764,Z 401.403,A -85,B 0,C 180,E1 -13680.002,E2 -13680.002} C_VEL
LIN {X 0,Y 346.834,Z 402.338,A -85,B 0,C 180,E1 -13681.163,E2 -13681.163} C_VEL
LIN {X 0,Y 347.002,Z 402.621,A -85,B 0,C 180,E1 -13682.323,E2 -13682.323} C_VEL
LIN {X 0,Y 347.305,Z 402.253,A -85,B 0,C 180,E1 -13683.482,E2 -13683.482} C_VEL
LIN {X 0,Y 347.78,Z 401.22,A -85,B 0,C 180,E1 -13684.638,E2 -13684.638} C_VEL
LIN {X 0,Y 348.675,Z 398.452,A -85,B 0,C 180,E1 -13686.366,E2 -13686.366} C_VEL
LIN {X 0,Y 349.653,Z 394.124,A -85,B 0,C 180,E1 -13688.09,E2 -13688.09} C_VEL
LIN {X 0,Y 350.89,Z 387.98,A -85,B 0,C 180,E1 -13689.804,E2 -13689.804} C_VEL
LIN {X 0,Y 352.122,Z 381.218,A -85,B 0,C 180,E1 -13691.223,E2 -13691.223} C_VEL
LIN {X 0,Y 353.417,Z 373.588,A -85,B 0,C 180,E1 -13692.491,E2 -13692.491} C_VEL
LIN {X 0,Y 354.51,Z 366.041,A -85,B 0,C 180,E1 -13693.502,E2 -13693.502} C_VEL
LIN {X 0,Y 353.826,Z 359.098,A -85,B 0,C 180,E1 -13694.427,E2 -13694.427} C_VEL
LIN {X 0,Y 351.173,Z 348.202,A -85,B 0,C 180,E1 -13695.8,E2 -13695.8} C_VEL
LIN {X 0,Y 348.789,Z 341.03,A -85,B 0,C 180,E1 -13696.688,E2 -13696.688} C_VEL
LIN {X 0,Y 349.367,Z 336.469,A -85,B 0,C 180,E1 -13699.999,E2 -13699.999} C_VEL
LIN {X 0,Y 350.161,Z 331.807,A -85,B 0,C 180,E1 -13703.668,E2 -13703.668} C_VEL
LIN {X 0,Y 351.094,Z 327.508,A -85,B 0,C 180,E1 -13707.414,E2 -13707.414} C_VEL
LIN {X 0,Y 351.912,Z 324.22,A -85,B 0,C 180,E1 -13710.823,E2 -13710.823} C_VEL
LIN {X 0,Y 352.147,Z 322.54,A -85,B 0,C 180,E1 -13713.047,E2 -13713.047} C_VEL
LIN {X 0,Y 352.172,Z 321.167,A -85,B 0,C 180,E1 -13715.363,E2 -13715.363} C_VEL
LIN {X 0,Y 352.18,Z 319.974,A -85,B 0,C 180,E1 -13718.897,E2 -13718.897} C_VEL
LIN {X 0,Y 352.329,Z 319.927,A -85,B 0,C 180,E1 -13722.434,E2 -13722.434} C_VEL
LIN {X 0,Y 352.704,Z 321.004,A -85,B 0,C 180,E1 -13725.837,E2 -13725.837} C_VEL
LIN {X 0,Y 353.29,Z 323.189,A -85,B 0,C 180,E1 -13729.109,E2 -13729.109} C_VEL
LIN {X 0,Y 354.028,Z 326.206,A -85,B 0,C 180,E1 -13732.019,E2 -13732.019} C_VEL
LIN {X 0,Y 354.915,Z 330.212,A -85,B 0,C 180,E1 -13734.952,E2 -13734.952} C_VEL
LIN {X 0,Y 355.833,Z 335.005,A -85,B 0,C 180,E1 -13737.773,E2 -13737.773} C_VEL
LIN {X 0,Y 355.912,Z 337.719,A -85,B 0,C 180,E1 -13739.109,E2 -13739.109} C_VEL
LIN {X 0,Y 354.118,Z 343.879,A -85,B 0,C 180,E1 -13741.555,E2 -13741.555} C_VEL
LIN {X 0,Y 351.674,Z 353.94,A -85,B 0,C 180,E1 -13745.186,E2 -13745.186} C_VEL
LIN {X 0,Y 350.112,Z 362.84,A -85,B 0,C 180,E1 -13748.123,E2 -13748.123} C_VEL
LIN {X 0,Y 352.632,Z 374.913,A -85,B 0,C 180,E1 -13748.958,E2 -13748.958} C_VEL
LIN {X 0,Y 353.923,Z 386.178,A -85,B 0,C 180,E1 -13749.811,E2 -13749.811} C_VEL
LIN {X 0,Y 353.907,Z 397.113,A -85,B 0,C 180,E1 -13750.722,E2 -13750.722} C_VEL
LIN {X 0,Y 353.148,Z 406.13,A -85,B 0,C 180,E1 -13751.583,E2 -13751.583} C_VEL
LIN {X 0,Y 351.328,Z 418.346,A -85,B 0,C 180,E1 -13752.989,E2 -13752.989} C_VEL
LIN {X 0,Y 349.979,Z 427.606,A -85,B 0,C 180,E1 -13754.33,E2 -13754.33} C_VEL
LIN {X 0,Y 348.638,Z 436.938,A -85,B 0,C 180,E1 -13756.001,E2 -13756.001} C_VEL
LIN {X 0,Y 347.733,Z 444.777,A -85,B 0,C 180,E1 -13757.748,E2 -13757.748} C_VEL
LIN {X 0,Y 346.915,Z 451.078,A -85,B 0,C 180,E1 -13759.495,E2 -13759.495} C_VEL
LIN {X 0,Y 346.567,Z 456.128,A -85,B 0,C 180,E1 -13761.252,E2 -13761.252} C_VEL
LIN {X 0,Y 346.437,Z 460.04,A -85,B 0,C 180,E1 -13763.009,E2 -13763.009} C_VEL
LIN {X 0,Y 346.421,Z 462.08,A -85,B 0,C 180,E1 -13764.178,E2 -13764.178} C_VEL
LIN {X 0,Y 346.45,Z 463.627,A -85,B 0,C 180,E1 -13765.346,E2 -13765.346} C_VEL
LIN {X 0,Y 346.56,Z 464.761,A -85,B 0,C 180,E1 -13766.512,E2 -13766.512} C_VEL
LIN {X 0,Y 346.689,Z 465.478,A -85,B 0,C 180,E1 -13767.676,E2 -13767.676} C_VEL
LIN {X 0,Y 346.743,Z 465.712,A -85,B 0,C 180,E1 -13768.839,E2 -13768.839} C_VEL
LIN {X 0,Y 346.71,Z 465.517,A -85,B 0,C 180,E1 -13770,E2 -13770} C_VEL
LIN {X 0,Y 346.75,Z 464.901,A -85,B 0,C 180,E1 -13771.161,E2 -13771.161} C_VEL
LIN {X 0,Y 346.851,Z 463.813,A -85,B 0,C 180,E1 -13772.323,E2 -13772.323} C_VEL
LIN {X 0,Y 346.701,Z 462.624,A -85,B 0,C 180,E1 -13773.487,E2 -13773.487} C_VEL
LIN {X 0,Y 346.607,Z 460.815,A -85,B 0,C 180,E1 -13774.652,E2 -13774.652} C_VEL
LIN {X 0,Y 346.687,Z 456.974,A -85,B 0,C 180,E1 -13776.278,E2 -13776.278} C_VEL
LIN {X 0,Y 346.696,Z 451.734,A -85,B 0,C 180,E1 -13777.865,E2 -13777.865} C_VEL
LIN {X 0,Y 346.82,Z 445.089,A -85,B 0,C 180,E1 -13779.624,E2 -13779.624} C_VEL
LIN {X 0,Y 347.238,Z 436.733,A -85,B 0,C 180,E1 -13781.381,E2 -13781.381} C_VEL
LIN {X 0,Y 347.795,Z 428.017,A -85,B 0,C 180,E1 -13782.843,E2 -13782.843} C_VEL
LIN {X 0,Y 348.312,Z 418.363,A -85,B 0,C 180,E1 -13784.16,E2 -13784.16} C_VEL
LIN {X 0,Y 349.026,Z 407.693,A -85,B 0,C 180,E1 -13785.325,E2 -13785.325} C_VEL
LIN {X 0,Y 349.75,Z 395.797,A -85,B 0,C 180,E1 -13786.339,E2 -13786.339} C_VEL
LIN {X 0,Y 349.129,Z 385.281,A -85,B 0,C 180,E1 -13787.046,E2 -13787.046} C_VEL
LIN {X 0,Y 348.224,Z 373.362,A -85,B 0,C 180,E1 -13787.644,E2 -13787.644} C_VEL
LIN {X 0,Y 347.78,Z 365.013,A -85,B 0,C 180,E1 -13787.947,E2 -13787.947} C_VEL
LIN {X 0,Y 349.222,Z 349.977,A -85,B 0,C 180,E1 -13792.481,E2 -13792.481} C_VEL
LIN {X 0,Y 351.203,Z 334.86,A -85,B 0,C 180,E1 -13797.081,E2 -13797.081} C_VEL
LIN {X 0,Y 352.52,Z 325.743,A -85,B 0,C 180,E1 -13799.895,E2 -13799.895} C_VEL
LIN {X 0,Y 351.982,Z 321.542,A -85,B 0,C 180,E1 -13801.275,E2 -13801.275} C_VEL
LIN {X 0,Y 349.692,Z 310.535,A -85,B 0,C 180,E1 -13805.058,E2 -13805.058} C_VEL
LIN {X 0,Y 347.829,Z 301.16,A -85,B 0,C 180,E1 -13808.454,E2 -13808.454} C_VEL
LIN {X 0,Y 347.756,Z 301.167,A -85,B 0,C 180,E1 -13811.83,E2 -13811.83} C_VEL
LIN {X 0,Y 347.711,Z 301.171,A -85,B 0,C 180,E1 -13815.026,E2 -13815.026} C_VEL
LIN {X 0,Y 347.756,Z 301.165,A -85,B 0,C 180,E1 -13818.397,E2 -13818.397} C_VEL
LIN {X 0,Y 347.792,Z 301.22,A -85,B 0,C 180,E1 -13820.933,E2 -13820.933} C_VEL
LIN {X 0,Y 349.167,Z 306.146,A -85,B 0,C 180,E1 -13824.287,E2 -13824.287} C_VEL
LIN {X 0,Y 350.321,Z 311.35,A -85,B 0,C 180,E1 -13827.415,E2 -13827.415} C_VEL
LIN {X 0,Y 350.994,Z 315.918,A -85,B 0,C 180,E1 -13829.96,E2 -13829.96} C_VEL
LIN {X 0,Y 350.667,Z 321.061,A -85,B 0,C 180,E1 -13832.549,E2 -13832.549} C_VEL
LIN {X 0,Y 350.11,Z 328.76,A -85,B 0,C 180,E1 -13836.328,E2 -13836.328} C_VEL
LIN {X 0,Y 349.73,Z 336.275,A -85,B 0,C 180,E1 -13840.023,E2 -13840.023} C_VEL
LIN {X 0,Y 349.355,Z 343.69,A -85,B 0,C 180,E1 -13843.641,E2 -13843.641} C_VEL
LIN {X 0,Y 349.26,Z 348.543,A -85,B 0,C 180,E1 -13845.935,E2 -13845.935} C_VEL
LIN {X 0,Y 351.67,Z 356.888,A -85,B 0,C 180,E1 -13846.712,E2 -13846.712} C_VEL
LIN {X 0,Y 352.748,Z 362.942,A -85,B 0,C 180,E1 -13847.339,E2 -13847.339} C_VEL
LIN {X 0,Y 351.988,Z 371.858,A -85,B 0,C 180,E1 -13848.287,E2 -13848.287} C_VEL
LIN {X 0,Y 351.092,Z 379.067,A -85,B 0,C 180,E1 -13849.29,E2 -13849.29} C_VEL
LIN {X 0,Y 350.28,Z 385.705,A -85,B 0,C 180,E1 -13850.471,E2 -13850.471} C_VEL
LIN {X 0,Y 349.668,Z 390.635,A -85,B 0,C 180,E1 -13851.62,E2 -13851.62} C_VEL
LIN {X 0,Y 348.842,Z 395.405,A -85,B 0,C 180,E1 -13853.056,E2 -13853.056} C_VEL
LIN {X 0,Y 348.3,Z 398.224,A -85,B 0,C 180,E1 -13854.208,E2 -13854.208} C_VEL
LIN {X 0,Y 347.762,Z 400.254,A -85,B 0,C 180,E1 -13855.362,E2 -13855.362} C_VEL
LIN {X 0,Y 347.272,Z 401.541,A -85,B 0,C 180,E1 -13856.518,E2 -13856.518} C_VEL
LIN {X 0,Y 346.974,Z 402.114,A -85,B 0,C 180,E1 -13857.677,E2 -13857.677} C_VEL
LIN {X 0,Y 346.814,Z 401.995,A -85,B 0,C 180,E1 -13858.837,E2 -13858.837} C_VEL
LIN {X 0,Y 346.751,Z 401.188,A -85,B 0,C 180,E1 -13859.998,E2 -13859.998} C_VEL
LIN {X 0,Y 346.73,Z 398.706,A -85,B 0,C 180,E1 -13861.741,E2 -13861.741} C_VEL
LIN {X 0,Y 346.871,Z 394.458,A -85,B 0,C 180,E1 -13863.483,E2 -13863.483} C_VEL
LIN {X 0,Y 347.126,Z 389.38,A -85,B 0,C 180,E1 -13864.935,E2 -13864.935} C_VEL
LIN {X 0,Y 347.342,Z 384.141,A -85,B 0,C 180,E1 -13866.096,E2 -13866.096} C_VEL
LIN {X 0,Y 347.504,Z 376.567,A -85,B 0,C 180,E1 -13867.394,E2 -13867.394} C_VEL
LIN {X 0,Y 347.715,Z 368.878,A -85,B 0,C 180,E1 -13868.425,E2 -13868.425} C_VEL
LIN {X 0,Y 347.924,Z 360.308,A -85,B 0,C 180,E1 -13869.298,E2 -13869.298} C_VEL
LIN {X 0,Y 348.081,Z 350.914,A -85,B 0,C 180,E1 -13870.027,E2 -13870.027} C_VEL
LIN {X 0,Y 347.233,Z 343.758,A -85,B 0,C 180,E1 -13870.457,E2 -13870.457} C_VEL
LIN {X 0,Y 347.326,Z 336.306,A -85,B 0,C 180,E1 -13873.769,E2 -13873.769} C_VEL
LIN {X 0,Y 347.345,Z 327.658,A -85,B 0,C 180,E1 -13877.666,E2 -13877.666} C_VEL
LIN {X 0,Y 347.483,Z 319.581,A -85,B 0,C 180,E1 -13881.348,E2 -13881.348} C_VEL
LIN {X 0,Y 347.657,Z 311.366,A -85,B 0,C 180,E1 -13885.118,E2 -13885.118} C_VEL
LIN {X 0,Y 347.776,Z 304.376,A -85,B 0,C 180,E1 -13888.351,E2 -13888.351} C_VEL
LIN {X 0,Y 347.903,Z 301.147,A -85,B 0,C 180,E1 -13889.815,E2 -13889.815} C_VEL
LIN {X 0,Y 347.739,Z 301.166,A -85,B 0,C 180,E1 -13894.462,E2 -13894.462} C_VEL
LIN {X 0,Y 347.757,Z 301.164,A -85,B 0,C 180,E1 -13897.985,E2 -13897.985} C_VEL
LIN {X 0,Y 347.737,Z 301.167,A -85,B 0,C 180,E1 -13901.83,E2 -13901.83} C_VEL
LIN {X 0,Y 347.698,Z 301.176,A -85,B 0,C 180,E1 -13905.025,E2 -13905.025} C_VEL
LIN {X 0,Y 347.743,Z 301.167,A -85,B 0,C 180,E1 -13908.396,E2 -13908.396} C_VEL
LIN {X 0,Y 347.769,Z 301.163,A -85,B 0,C 180,E1 -13912.009,E2 -13912.009} C_VEL
LIN {X 0,Y 347.735,Z 301.167,A -85,B 0,C 180,E1 -13915.535,E2 -13915.535} C_VEL
LIN {X 0,Y 347.755,Z 301.165,A -85,B 0,C 180,E1 -13919.652,E2 -13919.652} C_VEL
LIN {X 0,Y 347.842,Z 301.158,A -85,B 0,C 180,E1 -13922.743,E2 -13922.743} C_VEL
LIN {X 0,Y 347.778,Z 301.164,A -85,B 0,C 180,E1 -13926.161,E2 -13926.161} C_VEL
LIN {X 0,Y 347.806,Z 301.16,A -85,B 0,C 180,E1 -13929.909,E2 -13929.909} C_VEL
LIN {X 0,Y 347.855,Z 301.157,A -85,B 0,C 180,E1 -13932.359,E2 -13932.359} C_VEL
LIN {X 0,Y 347.886,Z 301.151,A -85,B 0,C 180,E1 -13935.97,E2 -13935.97} C_VEL
LIN {X 0,Y 347.884,Z 301.149,A -85,B 0,C 180,E1 -13939.524,E2 -13939.524} C_VEL
LIN {X 0,Y 348.044,Z 301.128,A -85,B 0,C 180,E1 -13943.041,E2 -13943.041} C_VEL
LIN {X 0,Y 348.177,Z 301.114,A -85,B 0,C 180,E1 -13947.686,E2 -13947.686} C_VEL
LIN {X 0,Y 348.103,Z 301.121,A -85,B 0,C 180,E1 -13951.157,E2 -13951.157} C_VEL
LIN {X 0,Y 348.177,Z 301.114,A -85,B 0,C 180,E1 -13952.314,E2 -13952.314} C_VEL
LIN {X 0,Y 348.044,Z 301.128,A -85,B 0,C 180,E1 -13956.959,E2 -13956.959} C_VEL
LIN {X 0,Y 347.884,Z 301.149,A -85,B 0,C 180,E1 -13960.476,E2 -13960.476} C_VEL
LIN {X 0,Y 347.887,Z 301.15,A -85,B 0,C 180,E1 -13964.15,E2 -13964.15} C_VEL
LIN {X 0,Y 347.88,Z 301.15,A -85,B 0,C 180,E1 -13968.291,E2 -13968.291} C_VEL
LIN {X 0,Y 347.778,Z 301.166,A -85,B 0,C 180,E1 -13971.636,E2 -13971.636} C_VEL
LIN {X 0,Y 347.802,Z 301.162,A -85,B 0,C 180,E1 -13975.109,E2 -13975.109} C_VEL
LIN {X 0,Y 347.802,Z 301.162,A -85,B 0,C 180,E1 -13977.695,E2 -13977.695} C_VEL
LIN {X 0,Y 347.755,Z 301.165,A -85,B 0,C 180,E1 -13980.348,E2 -13980.348} C_VEL
LIN {X 0,Y 347.735,Z 301.167,A -85,B 0,C 180,E1 -13984.465,E2 -13984.465} C_VEL
LIN {X 0,Y 347.769,Z 301.163,A -85,B 0,C 180,E1 -13987.991,E2 -13987.991} C_VEL
LIN {X 0,Y 347.743,Z 301.166,A -85,B 0,C 180,E1 -13991.832,E2 -13991.832} C_VEL
LIN {X 0,Y 347.698,Z 301.177,A -85,B 0,C 180,E1 -13995.028,E2 -13995.028} C_VEL
LIN {X 0,Y 347.734,Z 301.168,A -85,B 0,C 180,E1 -13998.401,E2 -13998.401} C_VEL
LIN {X 0,Y 347.75,Z 301.169,A -85,B 0,C 180,E1 -14002.68,E2 -14002.68} C_VEL
LIN {X 0,Y 347.743,Z 301.166,A -85,B 0,C 180,E1 -14005.958,E2 -14005.958} C_VEL
LIN {X 0,Y 347.99,Z 301.317,A -85,B 0,C 180,E1 -14008.708,E2 -14008.708} C_VEL
LIN {X 0,Y 347.432,Z 302.913,A -85,B 0,C 180,E1 -14009.638,E2 -14009.638} C_VEL
LIN {X 0,Y 344.515,Z 305.758,A -85,B 0,C 180,E1 -14011.136,E2 -14011.136} C_VEL
LIN {X 0,Y 341.933,Z 308.079,A -85,B 0,C 180,E1 -14012.346,E2 -14012.346} C_VEL
LIN {X 0,Y 340.778,Z 309.783,A -85,B 0,C 180,E1 -14013.289,E2 -14013.289} C_VEL
LIN {X 0,Y 340.666,Z 310.332,A -85,B 0,C 180,E1 -14013.611,E2 -14013.611} C_VEL
LIN {X 0,Y 340.321,Z 316.982,A -85,B 0,C 180,E1 -14017.541,E2 -14017.541} C_VEL
LIN {X 0,Y 340.089,Z 322.409,A -85,B 0,C 180,E1 -14020.694,E2 -14020.694} C_VEL
LIN {X 0,Y 339.823,Z 328.919,A -85,B 0,C 180,E1 -14024.405,E2 -14024.405} C_VEL
LIN {X 0,Y 339.676,Z 335.466,A -85,B 0,C 180,E1 -14028.061,E2 -14028.061} C_VEL
LIN {X 0,Y 339.685,Z 335.755,A -85,B 0,C 180,E1 -14028.213,E2 -14028.213} C_VEL
LIN {X 0,Y 340.844,Z 346.714,A -85,B 0,C 180,E1 -14028.931,E2 -14028.931} C_VEL
LIN {X 0,Y 341.596,Z 353.3,A -85,B 0,C 180,E1 -14029.481,E2 -14029.481} C_VEL
LIN {X 0,Y 341.146,Z 363.563,A -85,B 0,C 180,E1 -14030.516,E2 -14030.516} C_VEL
LIN {X 0,Y 340.797,Z 372.725,A -85,B 0,C 180,E1 -14031.702,E2 -14031.702} C_VEL
LIN {X 0,Y 340.519,Z 380.028,A -85,B 0,C 180,E1 -14032.888,E2 -14032.888} C_VEL
LIN {X 0,Y 340.217,Z 387.256,A -85,B 0,C 180,E1 -14034.371,E2 -14034.371} C_VEL
LIN {X 0,Y 339.993,Z 392.882,A -85,B 0,C 180,E1 -14035.853,E2 -14035.853} C_VEL
LIN {X 0,Y 339.699,Z 397.866,A -85,B 0,C 180,E1 -14037.63,E2 -14037.63} C_VEL
LIN {X 0,Y 339.651,Z 400.259,A -85,B 0,C 180,E1 -14038.816,E2 -14038.816} C_VEL
LIN {X 0,Y 339.715,Z 401.965,A -85,B 0,C 180,E1 -14040.002,E2 -14040.002} C_VEL
LIN {X 0,Y 339.787,Z 403.016,A -85,B 0,C 180,E1 -14041.187,E2 -14041.187} C_VEL
LIN {X 0,Y 339.962,Z 403.411,A -85,B 0,C 180,E1 -14042.371,E2 -14042.371} C_VEL
LIN {X 0,Y 340.276,Z 403.154,A -85,B 0,C 180,E1 -14043.554,E2 -14043.554} C_VEL
LIN {X 0,Y 340.778,Z 402.247,A -85,B 0,C 180,E1 -14044.733,E2 -14044.733} C_VEL
LIN {X 0,Y 341.744,Z 399.661,A -85,B 0,C 180,E1 -14046.496,E2 -14046.496} C_VEL
LIN {X 0,Y 342.763,Z 395.542,A -85,B 0,C 180,E1 -14048.253,E2 -14048.253} C_VEL
LIN {X 0,Y 344.073,Z 389.722,A -85,B 0,C 180,E1 -14050,E2 -14050} C_VEL
LIN {X 0,Y 345.387,Z 383.305,A -85,B 0,C 180,E1 -14051.445,E2 -14051.445} C_VEL
LIN {X 0,Y 346.907,Z 375.097,A -85,B 0,C 180,E1 -14052.878,E2 -14052.878} C_VEL
LIN {X 0,Y 348.108,Z 366.861,A -85,B 0,C 180,E1 -14054.022,E2 -14054.022} C_VEL
LIN {X 0,Y 346.898,Z 358.065,A -85,B 0,C 180,E1 -14055.272,E2 -14055.272} C_VEL
LIN {X 0,Y 344.46,Z 349.041,A -85,B 0,C 180,E1 -14056.475,E2 -14056.475} C_VEL
LIN {X 0,Y 341.996,Z 341.674,A -85,B 0,C 180,E1 -14057.414,E2 -14057.414} C_VEL
LIN {X 0,Y 342.555,Z 337.725,A -85,B 0,C 180,E1 -14060.414,E2 -14060.414} C_VEL
LIN {X 0,Y 343.412,Z 333.12,A -85,B 0,C 180,E1 -14064.163,E2 -14064.163} C_VEL
LIN {X 0,Y 344.432,Z 328.985,A -85,B 0,C 180,E1 -14067.991,E2 -14067.991} C_VEL
LIN {X 0,Y 345.165,Z 326.063,A -85,B 0,C 180,E1 -14071.221,E2 -14071.221} C_VEL
LIN {X 0,Y 345.407,Z 324.5,A -85,B 0,C 180,E1 -14073.464,E2 -14073.464} C_VEL
LIN {X 0,Y 345.454,Z 323.212,A -85,B 0,C 180,E1 -14076.157,E2 -14076.157} C_VEL
LIN {X 0,Y 345.525,Z 322.392,A -85,B 0,C 180,E1 -14079.383,E2 -14079.383} C_VEL
LIN {X 0,Y 345.726,Z 322.534,A -85,B 0,C 180,E1 -14082.961,E2 -14082.961} C_VEL
LIN {X 0,Y 346.136,Z 323.788,A -85,B 0,C 180,E1 -14086.343,E2 -14086.343} C_VEL
LIN {X 0,Y 346.757,Z 326.14,A -85,B 0,C 180,E1 -14089.566,E2 -14089.566} C_VEL
LIN {X 0,Y 347.548,Z 329.438,A -85,B 0,C 180,E1 -14092.652,E2 -14092.652} C_VEL
LIN {X 0,Y 348.505,Z 333.907,A -85,B 0,C 180,E1 -14095.774,E2 -14095.774} C_VEL
LIN {X 0,Y 349.119,Z 337.223,A -85,B 0,C 180,E1 -14097.726,E2 -14097.726} C_VEL
LIN {X 0,Y 349.251,Z 338.653,A -85,B 0,C 180,E1 -14098.453,E2 -14098.453} C_VEL
LIN {X 0,Y 348.588,Z 341.529,A -85,B 0,C 180,E1 -14099.733,E2 -14099.733} C_VEL
LIN {X 0,Y 345.853,Z 350.962,A -85,B 0,C 180,E1 -14103.397,E2 -14103.397} C_VEL
LIN {X 0,Y 343.495,Z 362.223,A -85,B 0,C 180,E1 -14107.382,E2 -14107.382} C_VEL
LIN {X 0,Y 346.364,Z 376.098,A -85,B 0,C 180,E1 -14108.422,E2 -14108.422} C_VEL
LIN {X 0,Y 347.529,Z 387.196,A -85,B 0,C 180,E1 -14109.326,E2 -14109.326} C_VEL
LIN {X 0,Y 347.361,Z 398.604,A -85,B 0,C 180,E1 -14110.344,E2 -14110.344} C_VEL
LIN {X 0,Y 346.307,Z 408.511,A -85,B 0,C 180,E1 -14111.359,E2 -14111.359} C_VEL
LIN {X 0,Y 344.594,Z 419,A -85,B 0,C 180,E1 -14112.646,E2 -14112.646} C_VEL
LIN {X 0,Y 342.967,Z 429.351,A -85,B 0,C 180,E1 -14114.245,E2 -14114.245} C_VEL
LIN {X 0,Y 341.556,Z 438.449,A -85,B 0,C 180,E1 -14116.009,E2 -14116.009} C_VEL
LIN {X 0,Y 340.598,Z 445.826,A -85,B 0,C 180,E1 -14117.79,E2 -14117.79} C_VEL
LIN {X 0,Y 339.879,Z 450.865,A -85,B 0,C 180,E1 -14119.275,E2 -14119.275} C_VEL
LIN {X 0,Y 339.51,Z 455.794,A -85,B 0,C 180,E1 -14121.068,E2 -14121.068} C_VEL
LIN {X 0,Y 339.359,Z 459.602,A -85,B 0,C 180,E1 -14122.862,E2 -14122.862} C_VEL
LIN {X 0,Y 339.351,Z 461.548,A -85,B 0,C 180,E1 -14124.056,E2 -14124.056} C_VEL
LIN {X 0,Y 339.377,Z 463.044,A -85,B 0,C 180,E1 -14125.248,E2 -14125.248} C_VEL
LIN {X 0,Y 339.467,Z 464.134,A -85,B 0,C 180,E1 -14126.439,E2 -14126.439} C_VEL
LIN {X 0,Y 339.617,Z 464.768,A -85,B 0,C 180,E1 -14127.628,E2 -14127.628} C_VEL
LIN {X 0,Y 339.696,Z 464.958,A -85,B 0,C 180,E1 -14128.815,E2 -14128.815} C_VEL
LIN {X 0,Y 339.665,Z 464.719,A -85,B 0,C 180,E1 -14130,E2 -14130} C_VEL
LIN {X 0,Y 339.784,Z 463.048,A -85,B 0,C 180,E1 -14132.371,E2 -14132.371} C_VEL
LIN {X 0,Y 339.602,Z 462.039,A -85,B 0,C 180,E1 -14133.559,E2 -14133.559} C_VEL
LIN {X 0,Y 339.525,Z 459.219,A -85,B 0,C 180,E1 -14135.345,E2 -14135.345} C_VEL
LIN {X 0,Y 339.607,Z 454.695,A -85,B 0,C 180,E1 -14137.133,E2 -14137.133} C_VEL
LIN {X 0,Y 339.667,Z 449.313,A -85,B 0,C 180,E1 -14138.627,E2 -14138.627} C_VEL
LIN {X 0,Y 339.969,Z 439.563,A -85,B 0,C 180,E1 -14140.723,E2 -14140.723} C_VEL
LIN {X 0,Y 340.415,Z 431.623,A -85,B 0,C 180,E1 -14142.217,E2 -14142.217} C_VEL
LIN {X 0,Y 341.03,Z 422.951,A -85,B 0,C 180,E1 -14143.557,E2 -14143.557} C_VEL
LIN {X 0,Y 341.633,Z 413.234,A -85,B 0,C 180,E1 -14144.785,E2 -14144.785} C_VEL
LIN {X 0,Y 342.356,Z 401.706,A -85,B 0,C 180,E1 -14145.936,E2 -14145.936} C_VEL
LIN {X 0,Y 342.61,Z 393.312,A -85,B 0,C 180,E1 -14146.613,E2 -14146.613} C_VEL
LIN {X 0,Y 341.589,Z 380.42,A -85,B 0,C 180,E1 -14147.435,E2 -14147.435} C_VEL
LIN {X 0,Y 340.849,Z 367.619,A -85,B 0,C 180,E1 -14147.997,E2 -14147.997} C_VEL
LIN {X 0,Y 340.742,Z 364.697,A -85,B 0,C 180,E1 -14148.115,E2 -14148.115} C_VEL
LIN {X 0,Y 342.45,Z 348.084,A -85,B 0,C 180,E1 -14153.27,E2 -14153.27} C_VEL
LIN {X 0,Y 344.384,Z 334.043,A -85,B 0,C 180,E1 -14157.663,E2 -14157.663} C_VEL
LIN {X 0,Y 345.49,Z 325.947,A -85,B 0,C 180,E1 -14160.23,E2 -14160.23} C_VEL
LIN {X 0,Y 344.23,Z 319.165,A -85,B 0,C 180,E1 -14162.553,E2 -14162.553} C_VEL
LIN {X 0,Y 342.152,Z 308.959,A -85,B 0,C 180,E1 -14166.196,E2 -14166.196} C_VEL
LIN {X 0,Y 340.756,Z 302.04,A -85,B 0,C 180,E1 -14168.843,E2 -14168.843} C_VEL
LIN {X 0,Y 340.681,Z 302.047,A -85,B 0,C 180,E1 -14172.904,E2 -14172.904} C_VEL
LIN {X 0,Y 340.681,Z 302.047,A -85,B 0,C 180,E1 -14177.095,E2 -14177.095} C_VEL
LIN {X 0,Y 340.718,Z 302.225,A -85,B 0,C 180,E1 -14178.985,E2 -14178.985} C_VEL
LIN {X 0,Y 341.824,Z 305.886,A -85,B 0,C 180,E1 -14181.915,E2 -14181.915} C_VEL
LIN {X 0,Y 343.023,Z 310.363,A -85,B 0,C 180,E1 -14185.039,E2 -14185.039} C_VEL
LIN {X 0,Y 343.934,Z 314.979,A -85,B 0,C 180,E1 -14187.906,E2 -14187.906} C_VEL
LIN {X 0,Y 344.348,Z 318.558,A -85,B 0,C 180,E1 -14189.996,E2 -14189.996} C_VEL
LIN {X 0,Y 343.944,Z 323.651,A -85,B 0,C 180,E1 -14192.627,E2 -14192.627} C_VEL
LIN {X 0,Y 343.449,Z 330.107,A -85,B 0,C 180,E1 -14195.84,E2 -14195.84} C_VEL
LIN {X 0,Y 342.995,Z 337.65,A -85,B 0,C 180,E1 -14199.613,E2 -14199.613} C_VEL
LIN {X 0,Y 342.56,Z 345.085,A -85,B 0,C 180,E1 -14203.307,E2 -14203.307} C_VEL
LIN {X 0,Y 342.485,Z 349.484,A -85,B 0,C 180,E1 -14205.398,E2 -14205.398} C_VEL
LIN {X 0,Y 345.203,Z 358.723,A -85,B 0,C 180,E1 -14206.308,E2 -14206.308} C_VEL
LIN {X 0,Y 346.22,Z 364.494,A -85,B 0,C 180,E1 -14206.947,E2 -14206.947} C_VEL
LIN {X 0,Y 345.45,Z 372.773,A -85,B 0,C 180,E1 -14207.863,E2 -14207.863} C_VEL
LIN {X 0,Y 344.43,Z 380.247,A -85,B 0,C 180,E1 -14208.94,E2 -14208.94} C_VEL
LIN {X 0,Y 343.675,Z 386.03,A -85,B 0,C 180,E1 -14209.988,E2 -14209.988} C_VEL
LIN {X 0,Y 342.809,Z 392.157,A -85,B 0,C 180,E1 -14211.451,E2 -14211.451} C_VEL
LIN {X 0,Y 341.927,Z 396.766,A -85,B 0,C 180,E1 -14212.915,E2 -14212.915} C_VEL
LIN {X 0,Y 341.336,Z 399.406,A -85,B 0,C 180,E1 -14214.09,E2 -14214.09} C_VEL
LIN {X 0,Y 340.758,Z 401.275,A -85,B 0,C 180,E1 -14215.266,E2 -14215.266} C_VEL
LIN {X 0,Y 340.244,Z 402.434,A -85,B 0,C 180,E1 -14216.446,E2 -14216.446} C_VEL
LIN {X 0,Y 339.936,Z 402.889,A -85,B 0,C 180,E1 -14217.629,E2 -14217.629} C_VEL
LIN {X 0,Y 339.768,Z 402.659,A -85,B 0,C 180,E1 -14218.813,E2 -14218.813} C_VEL
LIN {X 0,Y 339.685,Z 401.743,A -85,B 0,C 180,E1 -14219.998,E2 -14219.998} C_VEL
LIN {X 0,Y 339.653,Z 399.049,A -85,B 0,C 180,E1 -14221.777,E2 -14221.777} C_VEL
LIN {X 0,Y 339.787,Z 394.629,A -85,B 0,C 180,E1 -14223.556,E2 -14223.556} C_VEL
LIN {X 0,Y 340.053,Z 389.319,A -85,B 0,C 180,E1 -14225.038,E2 -14225.038} C_VEL
LIN {X 0,Y 340.334,Z 382.281,A -85,B 0,C 180,E1 -14226.52,E2 -14226.52} C_VEL
LIN {X 0,Y 340.439,Z 376.019,A -85,B 0,C 180,E1 -14227.549,E2 -14227.549} C_VEL
LIN {X 0,Y 340.644,Z 367.953,A -85,B 0,C 180,E1 -14228.601,E2 -14228.601} C_VEL
LIN {X 0,Y 340.919,Z 359.064,A -85,B 0,C 180,E1 -14229.491,E2 -14229.491} C_VEL
LIN {X 0,Y 340.965,Z 351.19,A -85,B 0,C 180,E1 -14230.089,E2 -14230.089} C_VEL
LIN {X 0,Y 340.166,Z 344.4,A -85,B 0,C 180,E1 -14230.489,E2 -14230.489} C_VEL
LIN {X 0,Y 340.266,Z 336.784,A -85,B 0,C 180,E1 -14233.889,E2 -14233.889} C_VEL
LIN {X 0,Y 340.295,Z 328.993,A -85,B 0,C 180,E1 -14237.424,E2 -14237.424} C_VEL
LIN {X 0,Y 340.429,Z 320.895,A -85,B 0,C 180,E1 -14241.134,E2 -14241.134} C_VEL
LIN {X 0,Y 340.594,Z 312.999,A -85,B 0,C 180,E1 -14244.78,E2 -14244.78} C_VEL
LIN {X 0,Y 340.732,Z 305.319,A -85,B 0,C 180,E1 -14248.318,E2 -14248.318} C_VEL
LIN {X 0,Y 340.869,Z 302.023,A -85,B 0,C 180,E1 -14249.894,E2 -14249.894} C_VEL
LIN {X 0,Y 340.718,Z 302.041,A -85,B 0,C 180,E1 -14254.403,E2 -14254.403} C_VEL
LIN {X 0,Y 340.713,Z 302.041,A -85,B 0,C 180,E1 -14258.228,E2 -14258.228} C_VEL
LIN {X 0,Y 340.687,Z 302.045,A -85,B 0,C 180,E1 -14262.043,E2 -14262.043} C_VEL
LIN {X 0,Y 340.644,Z 302.05,A -85,B 0,C 180,E1 -14266.225,E2 -14266.225} C_VEL
LIN {X 0,Y 340.68,Z 302.046,A -85,B 0,C 180,E1 -14269.752,E2 -14269.752} C_VEL
LIN {X 0,Y 340.698,Z 302.045,A -85,B 0,C 180,E1 -14273.257,E2 -14273.257} C_VEL
LIN {X 0,Y 340.683,Z 302.046,A -85,B 0,C 180,E1 -14276.152,E2 -14276.152} C_VEL
LIN {X 0,Y 340.765,Z 302.038,A -85,B 0,C 180,E1 -14280.331,E2 -14280.331} C_VEL
LIN {X 0,Y 340.795,Z 302.034,A -85,B 0,C 180,E1 -14283.019,E2 -14283.019} C_VEL
LIN {X 0,Y 340.718,Z 302.043,A -85,B 0,C 180,E1 -14286.926,E2 -14286.926} C_VEL
LIN {X 0,Y 340.784,Z 302.036,A -85,B 0,C 180,E1 -14290.733,E2 -14290.733} C_VEL
LIN {X 0,Y 340.775,Z 302.034,A -85,B 0,C 180,E1 -14293.218,E2 -14293.218} C_VEL
LIN {X 0,Y 340.832,Z 302.028,A -85,B 0,C 180,E1 -14296.89,E2 -14296.89} C_VEL
LIN {X 0,Y 340.869,Z 302.025,A -85,B 0,C 180,E1 -14300.506,E2 -14300.506} C_VEL
LIN {X 0,Y 340.99,Z 302.007,A -85,B 0,C 180,E1 -14302.896,E2 -14302.896} C_VEL
LIN {X 0,Y 340.805,Z 302.03,A -85,B 0,C 180,E1 -14305.268,E2 -14305.268} C_VEL
LIN {X 0,Y 341.114,Z 301.993,A -85,B 0,C 180,E1 -14307.638,E2 -14307.638} C_VEL
LIN {X 0,Y 341.075,Z 301.996,A -85,B 0,C 180,E1 -14311.181,E2 -14311.181} C_VEL
LIN {X 0,Y 341.114,Z 301.993,A -85,B 0,C 180,E1 -14312.362,E2 -14312.362} C_VEL
LIN {X 0,Y 341.005,Z 302.01,A -85,B 0,C 180,E1 -14315.915,E2 -14315.915} C_VEL
LIN {X 0,Y 340.951,Z 302.013,A -85,B 0,C 180,E1 -14318.357,E2 -14318.357} C_VEL
LIN {X 0,Y 340.837,Z 302.03,A -85,B 0,C 180,E1 -14321.9,E2 -14321.9} C_VEL
LIN {X 0,Y 340.808,Z 302.035,A -85,B 0,C 180,E1 -14325.55,E2 -14325.55} C_VEL
LIN {X 0,Y 340.827,Z 302.028,A -85,B 0,C 180,E1 -14328.468,E2 -14328.468} C_VEL
LIN {X 0,Y 340.743,Z 302.041,A -85,B 0,C 180,E1 -14331.858,E2 -14331.858} C_VEL
LIN {X 0,Y 340.762,Z 302.039,A -85,B 0,C 180,E1 -14335.665,E2 -14335.665} C_VEL
LIN {X 0,Y 340.732,Z 302.039,A -85,B 0,C 180,E1 -14338.321,E2 -14338.321} C_VEL
LIN {X 0,Y 340.695,Z 302.047,A -85,B 0,C 180,E1 -14341.045,E2 -14341.045} C_VEL
LIN {X 0,Y 340.71,Z 302.047,A -85,B 0,C 180,E1 -14345.28,E2 -14345.28} C_VEL
LIN {X 0,Y 340.704,Z 302.043,A -85,B 0,C 180,E1 -14348.388,E2 -14348.388} C_VEL
LIN {X 0,Y 340.691,Z 302.044,A -85,B 0,C 180,E1 -14352.047,E2 -14352.047} C_VEL
LIN {X 0,Y 340.644,Z 302.05,A -85,B 0,C 180,E1 -14356.229,E2 -14356.229} C_VEL
LIN {X 0,Y 340.664,Z 302.051,A -85,B 0,C 180,E1 -14358.69,E2 -14358.69} C_VEL
LIN {X 0,Y 340.712,Z 302.041,A -85,B 0,C 180,E1 -14361.772,E2 -14361.772} C_VEL
LIN {X 0,Y 340.718,Z 302.041,A -85,B 0,C 180,E1 -14365.597,E2 -14365.597} C_VEL
LIN {X 0,Y 340.935,Z 302.173,A -85,B 0,C 180,E1 -14368.636,E2 -14368.636} C_VEL
LIN {X 0,Y 341.036,Z 304.936,A -85,B 0,C 180,E1 -14370.36,E2 -14370.36} C_VEL
LIN {X 0,Y 340.666,Z 310.332,A -85,B 0,C 180,E1 -14373.611,E2 -14373.611} C_VEL
LIN {X 0,Y 339.922,Z 312.001,A -85,B 0,C 180,E1 -14374.556,E2 -14374.556} C_VEL
LIN {X 0,Y 336.923,Z 314.899,A -85,B 0,C 180,E1 -14376.079,E2 -14376.079} C_VEL
LIN {X 0,Y 334.386,Z 317.241,A -85,B 0,C 180,E1 -14377.311,E2 -14377.311} C_VEL
LIN {X 0,Y 333.267,Z 318.971,A -85,B 0,C 180,E1 -14378.271,E2 -14378.271} C_VEL
LIN {X 0,Y 333.158,Z 319.533,A -85,B 0,C 180,E1 -14378.598,E2 -14378.598} C_VEL
LIN {X 0,Y 332.939,Z 324.982,A -85,B 0,C 180,E1 -14381.788,E2 -14381.788} C_VEL
LIN {X 0,Y 332.692,Z 331.125,A -85,B 0,C 180,E1 -14385.317,E2 -14385.317} C_VEL
LIN {X 0,Y 332.601,Z 336.009,A -85,B 0,C 180,E1 -14388.074,E2 -14388.074} C_VEL
LIN {X 0,Y 333.908,Z 348.331,A -85,B 0,C 180,E1 -14388.929,E2 -14388.929} C_VEL
LIN {X 0,Y 334.533,Z 353.887,A -85,B 0,C 180,E1 -14389.409,E2 -14389.409} C_VEL
LIN {X 0,Y 334.064,Z 364.068,A -85,B 0,C 180,E1 -14390.465,E2 -14390.465} C_VEL
LIN {X 0,Y 333.759,Z 372.186,A -85,B 0,C 180,E1 -14391.525,E2 -14391.525} C_VEL
LIN {X 0,Y 333.438,Z 379.694,A -85,B 0,C 180,E1 -14392.736,E2 -14392.736} C_VEL
LIN {X 0,Y 333.158,Z 387.167,A -85,B 0,C 180,E1 -14394.251,E2 -14394.251} C_VEL
LIN {X 0,Y 332.911,Z 392.972,A -85,B 0,C 180,E1 -14395.764,E2 -14395.764} C_VEL
LIN {X 0,Y 332.639,Z 398.173,A -85,B 0,C 180,E1 -14397.58,E2 -14397.58} C_VEL
LIN {X 0,Y 332.578,Z 400.687,A -85,B 0,C 180,E1 -14398.791,E2 -14398.791} C_VEL
LIN {X 0,Y 332.635,Z 402.498,A -85,B 0,C 180,E1 -14400.002,E2 -14400.002} C_VEL
LIN {X 0,Y 332.741,Z 403.653,A -85,B 0,C 180,E1 -14401.212,E2 -14401.212} C_VEL
LIN {X 0,Y 332.923,Z 404.163,A -85,B 0,C 180,E1 -14402.421,E2 -14402.421} C_VEL
LIN {X 0,Y 333.248,Z 404.034,A -85,B 0,C 180,E1 -14403.629,E2 -14403.629} C_VEL
LIN {X 0,Y 333.775,Z 403.259,A -85,B 0,C 180,E1 -14404.833,E2 -14404.833} C_VEL
LIN {X 0,Y 334.81,Z 400.875,A -85,B 0,C 180,E1 -14406.631,E2 -14406.631} C_VEL
LIN {X 0,Y 335.9,Z 397.03,A -85,B 0,C 180,E1 -14408.423,E2 -14408.423} C_VEL
LIN {X 0,Y 337.278,Z 391.483,A -85,B 0,C 180,E1 -14410.203,E2 -14410.203} C_VEL
LIN {X 0,Y 338.668,Z 385.348,A -85,B 0,C 180,E1 -14411.675,E2 -14411.675} C_VEL
LIN {X 0,Y 340.275,Z 377.555,A -85,B 0,C 180,E1 -14413.133,E2 -14413.133} C_VEL
LIN {X 0,Y 341.722,Z 368.466,A -85,B 0,C 180,E1 -14414.489,E2 -14414.489} C_VEL
LIN {X 0,Y 340.61,Z 360.268,A -85,B 0,C 180,E1 -14415.721,E2 -14415.721} C_VEL
LIN {X 0,Y 338.186,Z 350.918,A -85,B 0,C 180,E1 -14417.069,E2 -14417.069} C_VEL
LIN {X 0,Y 335.229,Z 342.293,A -85,B 0,C 180,E1 -14418.243,E2 -14418.243} C_VEL
LIN {X 0,Y 336.032,Z 337.457,A -85,B 0,C 180,E1 -14422.116,E2 -14422.116} C_VEL
LIN {X 0,Y 337.03,Z 333.098,A -85,B 0,C 180,E1 -14425.972,E2 -14425.972} C_VEL
LIN {X 0,Y 337.914,Z 330.016,A -85,B 0,C 180,E1 -14429.129,E2 -14429.129} C_VEL
LIN {X 0,Y 338.467,Z 327.963,A -85,B 0,C 180,E1 -14431.643,E2 -14431.643} C_VEL
LIN {X 0,Y 338.693,Z 326.472,A -85,B 0,C 180,E1 -14434.075,E2 -14434.075} C_VEL
LIN {X 0,Y 338.75,Z 325.302,A -85,B 0,C 180,E1 -14436.99,E2 -14436.99} C_VEL
LIN {X 0,Y 338.861,Z 324.78,A -85,B 0,C 180,E1 -14440.013,E2 -14440.013} C_VEL
LIN {X 0,Y 339.105,Z 325.084,A -85,B 0,C 180,E1 -14443.153,E2 -14443.153} C_VEL
LIN {X 0,Y 339.55,Z 326.4,A -85,B 0,C 180,E1 -14446.423,E2 -14446.423} C_VEL
LIN {X 0,Y 340.203,Z 328.962,A -85,B 0,C 180,E1 -14449.851,E2 -14449.851} C_VEL
LIN {X 0,Y 340.676,Z 330.929,A -85,B 0,C 180,E1 -14451.765,E2 -14451.765} C_VEL
LIN {X 0,Y 341.532,Z 334.852,A -85,B 0,C 180,E1 -14454.818,E2 -14454.818} C_VEL
LIN {X 0,Y 342.422,Z 339.637,A -85,B 0,C 180,E1 -14457.748,E2 -14457.748} C_VEL
LIN {X 0,Y 342.472,Z 340.964,A -85,B 0,C 180,E1 -14458.446,E2 -14458.446} C_VEL
LIN {X 0,Y 341.17,Z 345.371,A -85,B 0,C 180,E1 -14460.37,E2 -14460.37} C_VEL
LIN {X 0,Y 338.38,Z 355.04,A -85,B 0,C 180,E1 -14464.141,E2 -14464.141} C_VEL
LIN {X 0,Y 336.978,Z 361.785,A -85,B 0,C 180,E1 -14466.589,E2 -14466.589} C_VEL
LIN {X 0,Y 339.954,Z 376.118,A -85,B 0,C 180,E1 -14467.755,E2 -14467.755} C_VEL
LIN {X 0,Y 341.154,Z 387.186,A -85,B 0,C 180,E1 -14468.722,E2 -14468.722} C_VEL
LIN {X 0,Y 340.966,Z 398.693,A -85,B 0,C 180,E1 -14469.803,E2 -14469.803} C_VEL
LIN {X 0,Y 339.868,Z 408.381,A -85,B 0,C 180,E1 -14470.836,E2 -14470.836} C_VEL
LIN {X 0,Y 338.055,Z 418.687,A -85,B 0,C 180,E1 -14472.143,E2 -14472.143} C_VEL
LIN {X 0,Y 336.397,Z 428.063,A -85,B 0,C 180,E1 -14473.618,E2 -14473.618} C_VEL
LIN {X 0,Y 334.862,Z 437.242,A -85,B 0,C 180,E1 -14475.413,E2 -14475.413} C_VEL
LIN {X 0,Y 333.822,Z 444.662,A -85,B 0,C 180,E1 -14477.229,E2 -14477.229} C_VEL
LIN {X 0,Y 332.858,Z 450.69,A -85,B 0,C 180,E1 -14479.046,E2 -14479.046} C_VEL
LIN {X 0,Y 332.47,Z 455.475,A -85,B 0,C 180,E1 -14480.878,E2 -14480.878} C_VEL
LIN {X 0,Y 332.282,Z 459.158,A -85,B 0,C 180,E1 -14482.709,E2 -14482.709} C_VEL
LIN {X 0,Y 332.273,Z 461.022,A -85,B 0,C 180,E1 -14483.929,E2 -14483.929} C_VEL
LIN {X 0,Y 332.306,Z 462.471,A -85,B 0,C 180,E1 -14485.147,E2 -14485.147} C_VEL
LIN {X 0,Y 332.377,Z 463.486,A -85,B 0,C 180,E1 -14486.363,E2 -14486.363} C_VEL
LIN {X 0,Y 332.546,Z 464.05,A -85,B 0,C 180,E1 -14487.577,E2 -14487.577} C_VEL
LIN {X 0,Y 332.65,Z 464.197,A -85,B 0,C 180,E1 -14488.789,E2 -14488.789} C_VEL
LIN {X 0,Y 332.621,Z 463.888,A -85,B 0,C 180,E1 -14490,E2 -14490} C_VEL
LIN {X 0,Y 332.702,Z 462.372,A -85,B 0,C 180,E1 -14492.421,E2 -14492.421} C_VEL
LIN {X 0,Y 332.504,Z 461.482,A -85,B 0,C 180,E1 -14493.636,E2 -14493.636} C_VEL
LIN {X 0,Y 332.431,Z 458.873,A -85,B 0,C 180,E1 -14495.459,E2 -14495.459} C_VEL
LIN {X 0,Y 332.501,Z 456.448,A -85,B 0,C 180,E1 -14496.565,E2 -14496.565} C_VEL
LIN {X 0,Y 332.564,Z 451.592,A -85,B 0,C 180,E1 -14498.201,E2 -14498.201} C_VEL
LIN {X 0,Y 332.725,Z 445.596,A -85,B 0,C 180,E1 -14499.729,E2 -14499.729} C_VEL
LIN {X 0,Y 332.948,Z 439.449,A -85,B 0,C 180,E1 -14500.951,E2 -14500.951} C_VEL
LIN {X 0,Y 333.962,Z 421.845,A -85,B 0,C 180,E1 -14503.695,E2 -14503.695} C_VEL
LIN {X 0,Y 334.624,Z 411.979,A -85,B 0,C 180,E1 -14504.952,E2 -14504.952} C_VEL
LIN {X 0,Y 335.367,Z 400.349,A -85,B 0,C 180,E1 -14506.121,E2 -14506.121} C_VEL
LIN {X 0,Y 335.485,Z 392.763,A -85,B 0,C 180,E1 -14506.741,E2 -14506.741} C_VEL
LIN {X 0,Y 334.474,Z 379.856,A -85,B 0,C 180,E1 -14507.581,E2 -14507.581} C_VEL
LIN {X 0,Y 333.854,Z 367.92,A -85,B 0,C 180,E1 -14508.169,E2 -14508.169} C_VEL
LIN {X 0,Y 333.869,Z 362.364,A -85,B 0,C 180,E1 -14508.923,E2 -14508.923} C_VEL
LIN {X 0,Y 335.437,Z 348.145,A -85,B 0,C 180,E1 -14513.459,E2 -14513.459} C_VEL
LIN {X 0,Y 337.434,Z 334.192,A -85,B 0,C 180,E1 -14517.945,E2 -14517.945} C_VEL
LIN {X 0,Y 338.49,Z 327.16,A -85,B 0,C 180,E1 -14520.232,E2 -14520.232} C_VEL
LIN {X 0,Y 337.107,Z 319.767,A -85,B 0,C 180,E1 -14522.823,E2 -14522.823} C_VEL
LIN {X 0,Y 335.053,Z 309.725,A -85,B 0,C 180,E1 -14526.501,E2 -14526.501} C_VEL
LIN {X 0,Y 333.701,Z 302.916,A -85,B 0,C 180,E1 -14529.185,E2 -14529.185} C_VEL
LIN {X 0,Y 333.638,Z 302.926,A -85,B 0,C 180,E1 -14532.499,E2 -14532.499} C_VEL
LIN {X 0,Y 333.628,Z 303.119,A -85,B 0,C 180,E1 -14535.959,E2 -14535.959} C_VEL
LIN {X 0,Y 334.652,Z 306.264,A -85,B 0,C 180,E1 -14539.379,E2 -14539.379} C_VEL
LIN {X 0,Y 335.811,Z 310.188,A -85,B 0,C 180,E1 -14542.682,E2 -14542.682} C_VEL
LIN {X 0,Y 336.479,Z 312.708,A -85,B 0,C 180,E1 -14544.547,E2 -14544.547} C_VEL
LIN {X 0,Y 337.246,Z 316.734,A -85,B 0,C 180,E1 -14547.191,E2 -14547.191} C_VEL
LIN {X 0,Y 337.771,Z 320.271,A -85,B 0,C 180,E1 -14549.35,E2 -14549.35} C_VEL
LIN {X 0,Y 337.517,Z 323.911,A -85,B 0,C 180,E1 -14551.384,E2 -14551.384} C_VEL
LIN {X 0,Y 336.811,Z 331.58,A -85,B 0,C 180,E1 -14555.333,E2 -14555.333} C_VEL
LIN {X 0,Y 336.256,Z 339.069,A -85,B 0,C 180,E1 -14559.186,E2 -14559.186} C_VEL
LIN {X 0,Y 335.785,Z 346.516,A -85,B 0,C 180,E1 -14562.96,E2 -14562.96} C_VEL
LIN {X 0,Y 335.672,Z 350.313,A -85,B 0,C 180,E1 -14564.792,E2 -14564.792} C_VEL
LIN {X 0,Y 338.403,Z 359.099,A -85,B 0,C 180,E1 -14565.721,E2 -14565.721} C_VEL
LIN {X 0,Y 339.709,Z 365.751,A -85,B 0,C 180,E1 -14566.496,E2 -14566.496} C_VEL
LIN {X 0,Y 338.911,Z 374.298,A -85,B 0,C 180,E1 -14567.482,E2 -14567.482} C_VEL
LIN {X 0,Y 337.812,Z 381.743,A -85,B 0,C 180,E1 -14568.599,E2 -14568.599} C_VEL
LIN {X 0,Y 336.899,Z 387.914,A -85,B 0,C 180,E1 -14569.785,E2 -14569.785} C_VEL
LIN {X 0,Y 335.946,Z 393.712,A -85,B 0,C 180,E1 -14571.275,E2 -14571.275} C_VEL
LIN {X 0,Y 335,Z 398.054,A -85,B 0,C 180,E1 -14572.767,E2 -14572.767} C_VEL
LIN {X 0,Y 334.365,Z 400.552,A -85,B 0,C 180,E1 -14573.966,E2 -14573.966} C_VEL
LIN {X 0,Y 333.756,Z 402.303,A -85,B 0,C 180,E1 -14575.167,E2 -14575.167} C_VEL
LIN {X 0,Y 333.218,Z 403.344,A -85,B 0,C 180,E1 -14576.371,E2 -14576.371} C_VEL
LIN {X 0,Y 332.899,Z 403.678,A -85,B 0,C 180,E1 -14577.579,E2 -14577.579} C_VEL
LIN {X 0,Y 332.723,Z 403.324,A -85,B 0,C 180,E1 -14578.788,E2 -14578.788} C_VEL
LIN {X 0,Y 332.606,Z 402.289,A -85,B 0,C 180,E1 -14579.998,E2 -14579.998} C_VEL
LIN {X 0,Y 332.553,Z 400.559,A -85,B 0,C 180,E1 -14581.209,E2 -14581.209} C_VEL
LIN {X 0,Y 332.64,Z 398.073,A -85,B 0,C 180,E1 -14582.42,E2 -14582.42} C_VEL
LIN {X 0,Y 332.86,Z 392.733,A -85,B 0,C 180,E1 -14584.236,E2 -14584.236} C_VEL
LIN {X 0,Y 333.11,Z 386.536,A -85,B 0,C 180,E1 -14585.75,E2 -14585.75} C_VEL
LIN {X 0,Y 333.302,Z 380.197,A -85,B 0,C 180,E1 -14586.962,E2 -14586.962} C_VEL
LIN {X 0,Y 333.487,Z 372.164,A -85,B 0,C 180,E1 -14588.146,E2 -14588.146} C_VEL
LIN {X 0,Y 333.745,Z 364.08,A -85,B 0,C 180,E1 -14589.085,E2 -14589.085} C_VEL
LIN {X 0,Y 333.92,Z 355.419,A -85,B 0,C 180,E1 -14589.845,E2 -14589.845} C_VEL
LIN {X 0,Y 333.803,Z 351.096,A -85,B 0,C 180,E1 -14590.154,E2 -14590.154} C_VEL
LIN {X 0,Y 333.102,Z 344.927,A -85,B 0,C 180,E1 -14590.56,E2 -14590.56} C_VEL
LIN {X 0,Y 333.221,Z 337.218,A -85,B 0,C 180,E1 -14594.024,E2 -14594.024} C_VEL
LIN {X 0,Y 333.261,Z 329.001,A -85,B 0,C 180,E1 -14597.773,E2 -14597.773} C_VEL
LIN {X 0,Y 333.391,Z 320.986,A -85,B 0,C 180,E1 -14601.47,E2 -14601.47} C_VEL
LIN {X 0,Y 333.548,Z 313.338,A -85,B 0,C 180,E1 -14605.037,E2 -14605.037} C_VEL
LIN {X 0,Y 333.695,Z 306.217,A -85,B 0,C 180,E1 -14608.318,E2 -14608.318} C_VEL
LIN {X 0,Y 333.836,Z 302.899,A -85,B 0,C 180,E1 -14609.969,E2 -14609.969} C_VEL
LIN {X 0,Y 333.68,Z 302.919,A -85,B 0,C 180,E1 -14614.772,E2 -14614.772} C_VEL
LIN {X 0,Y 333.637,Z 302.924,A -85,B 0,C 180,E1 -14617.651,E2 -14617.651} C_VEL
LIN {X 0,Y 333.597,Z 302.931,A -85,B 0,C 180,E1 -14620.772,E2 -14620.772} C_VEL
LIN {X 0,Y 333.586,Z 302.93,A -85,B 0,C 180,E1 -14624.249,E2 -14624.249} C_VEL
LIN {X 0,Y 333.634,Z 302.924,A -85,B 0,C 180,E1 -14627.617,E2 -14627.617} C_VEL
LIN {X 0,Y 333.646,Z 302.924,A -85,B 0,C 180,E1 -14631.2,E2 -14631.2} C_VEL
LIN {X 0,Y 333.668,Z 302.919,A -85,B 0,C 180,E1 -14633.86,E2 -14633.86} C_VEL
LIN {X 0,Y 333.634,Z 302.924,A -85,B 0,C 180,E1 -14637.412,E2 -14637.412} C_VEL
LIN {X 0,Y 333.702,Z 302.917,A -85,B 0,C 180,E1 -14641.027,E2 -14641.027} C_VEL
LIN {X 0,Y 333.726,Z 302.912,A -85,B 0,C 180,E1 -14643.753,E2 -14643.753} C_VEL
LIN {X 0,Y 333.709,Z 302.915,A -85,B 0,C 180,E1 -14647.913,E2 -14647.913} C_VEL
LIN {X 0,Y 333.783,Z 302.905,A -85,B 0,C 180,E1 -14651.589,E2 -14651.589} C_VEL
LIN {X 0,Y 333.797,Z 302.903,A -85,B 0,C 180,E1 -14655.576,E2 -14655.576} C_VEL
LIN {X 0,Y 333.805,Z 302.902,A -85,B 0,C 180,E1 -14659.077,E2 -14659.077} C_VEL
LIN {X 0,Y 333.945,Z 302.885,A -85,B 0,C 180,E1 -14662.746,E2 -14662.746} C_VEL
LIN {X 0,Y 333.771,Z 302.906,A -85,B 0,C 180,E1 -14665.169,E2 -14665.169} C_VEL
LIN {X 0,Y 334.055,Z 302.872,A -85,B 0,C 180,E1 -14667.588,E2 -14667.588} C_VEL
LIN {X 0,Y 334.045,Z 302.872,A -85,B 0,C 180,E1 -14671.206,E2 -14671.206} C_VEL
LIN {X 0,Y 334.055,Z 302.872,A -85,B 0,C 180,E1 -14672.412,E2 -14672.412} C_VEL
LIN {X 0,Y 333.978,Z 302.884,A -85,B 0,C 180,E1 -14676.04,E2 -14676.04} C_VEL
LIN {X 0,Y 333.808,Z 302.906,A -85,B 0,C 180,E1 -14679.697,E2 -14679.697} C_VEL
LIN {X 0,Y 333.785,Z 302.907,A -85,B 0,C 180,E1 -14683.392,E2 -14683.392} C_VEL
LIN {X 0,Y 333.735,Z 302.912,A -85,B 0,C 180,E1 -14687.147,E2 -14687.147} C_VEL
LIN {X 0,Y 333.731,Z 302.916,A -85,B 0,C 180,E1 -14689.691,E2 -14689.691} C_VEL
LIN {X 0,Y 333.682,Z 302.918,A -85,B 0,C 180,E1 -14692.279,E2 -14692.279} C_VEL
LIN {X 0,Y 333.726,Z 302.912,A -85,B 0,C 180,E1 -14696.247,E2 -14696.247} C_VEL
LIN {X 0,Y 333.702,Z 302.917,A -85,B 0,C 180,E1 -14698.973,E2 -14698.973} C_VEL
LIN {X 0,Y 333.634,Z 302.924,A -85,B 0,C 180,E1 -14702.588,E2 -14702.588} C_VEL
LIN {X 0,Y 333.668,Z 302.919,A -85,B 0,C 180,E1 -14706.14,E2 -14706.14} C_VEL
LIN {X 0,Y 333.639,Z 302.928,A -85,B 0,C 180,E1 -14709.194,E2 -14709.194} C_VEL
LIN {X 0,Y 333.625,Z 302.926,A -85,B 0,C 180,E1 -14712.501,E2 -14712.501} C_VEL
LIN {X 0,Y 333.589,Z 302.929,A -85,B 0,C 180,E1 -14715.956,E2 -14715.956} C_VEL
LIN {X 0,Y 333.596,Z 302.93,A -85,B 0,C 180,E1 -14719.326,E2 -14719.326} C_VEL
LIN {X 0,Y 333.656,Z 302.923,A -85,B 0,C 180,E1 -14723.17,E2 -14723.17} C_VEL
LIN {X 0,Y 333.668,Z 302.924,A -85,B 0,C 180,E1 -14726.797,E2 -14726.797} C_VEL
LIN {X 0,Y 333.863,Z 302.99,A -85,B 0,C 180,E1 -14728.541,E2 -14728.541} C_VEL
LIN {X 0,Y 333.992,Z 305.88,A -85,B 0,C 180,E1 -14730.366,E2 -14730.366} C_VEL
LIN {X 0,Y 333.618,Z 311.419,A -85,B 0,C 180,E1 -14733.746,E2 -14733.746} C_VEL
LIN {X 0,Y 333.261,Z 318,A -85,B 0,C 180,E1 -14737.693,E2 -14737.693} C_VEL
LIN {X 0,Y 333.158,Z 319.533,A -85,B 0,C 180,E1 -14738.598,E2 -14738.598} C_VEL
LIN {X 0,Y 332.42,Z 321.241,A -85,B 0,C 180,E1 -14739.562,E2 -14739.562} C_VEL
LIN {X 0,Y 329.447,Z 324.177,A -85,B 0,C 180,E1 -14741.119,E2 -14741.119} C_VEL
LIN {X 0,Y 326.934,Z 326.547,A -85,B 0,C 180,E1 -14742.378,E2 -14742.378} C_VEL
LIN {X 0,Y 325.829,Z 328.307,A -85,B 0,C 180,E1 -14743.359,E2 -14743.359} C_VEL
LIN {X 0,Y 325.724,Z 328.884,A -85,B 0,C 180,E1 -14743.692,E2 -14743.692} C_VEL
LIN {X 0,Y 325.553,Z 335.56,A -85,B 0,C 180,E1 -14747.535,E2 -14747.535} C_VEL
LIN {X 0,Y 325.529,Z 336.324,A -85,B 0,C 180,E1 -14747.969,E2 -14747.969} C_VEL
LIN {X 0,Y 326.822,Z 348.699,A -85,B 0,C 180,E1 -14748.843,E2 -14748.843} C_VEL
LIN {X 0,Y 327.457,Z 354.265,A -85,B 0,C 180,E1 -14749.334,E2 -14749.334} C_VEL
LIN {X 0,Y 326.983,Z 364.474,A -85,B 0,C 180,E1 -14750.413,E2 -14750.413} C_VEL
LIN {X 0,Y 326.627,Z 373.485,A -85,B 0,C 180,E1 -14751.626,E2 -14751.626} C_VEL
LIN {X 0,Y 326.306,Z 381.015,A -85,B 0,C 180,E1 -14752.888,E2 -14752.888} C_VEL
LIN {X 0,Y 326.03,Z 388.347,A -85,B 0,C 180,E1 -14754.435,E2 -14754.435} C_VEL
LIN {X 0,Y 325.812,Z 393.016,A -85,B 0,C 180,E1 -14755.672,E2 -14755.672} C_VEL
LIN {X 0,Y 325.562,Z 398.387,A -85,B 0,C 180,E1 -14757.527,E2 -14757.527} C_VEL
LIN {X 0,Y 325.508,Z 401.025,A -85,B 0,C 180,E1 -14758.764,E2 -14758.764} C_VEL
LIN {X 0,Y 325.558,Z 402.971,A -85,B 0,C 180,E1 -14760.002,E2 -14760.002} C_VEL
LIN {X 0,Y 325.697,Z 404.259,A -85,B 0,C 180,E1 -14761.238,E2 -14761.238} C_VEL
LIN {X 0,Y 325.886,Z 404.908,A -85,B 0,C 180,E1 -14762.474,E2 -14762.474} C_VEL
LIN {X 0,Y 326.221,Z 404.915,A -85,B 0,C 180,E1 -14763.707,E2 -14763.707} C_VEL
LIN {X 0,Y 326.775,Z 404.285,A -85,B 0,C 180,E1 -14764.937,E2 -14764.937} C_VEL
LIN {X 0,Y 327.419,Z 403.018,A -85,B 0,C 180,E1 -14766.163,E2 -14766.163} C_VEL
LIN {X 0,Y 328.644,Z 399.871,A -85,B 0,C 180,E1 -14767.992,E2 -14767.992} C_VEL
LIN {X 0,Y 330.001,Z 395.164,A -85,B 0,C 180,E1 -14769.811,E2 -14769.811} C_VEL
LIN {X 0,Y 331.595,Z 388.739,A -85,B 0,C 180,E1 -14771.617,E2 -14771.617} C_VEL
LIN {X 0,Y 333.269,Z 381.701,A -85,B 0,C 180,E1 -14773.104,E2 -14773.104} C_VEL
LIN {X 0,Y 335.071,Z 372.731,A -85,B 0,C 180,E1 -14774.579,E2 -14774.579} C_VEL
LIN {X 0,Y 335.319,Z 369.648,A -85,B 0,C 180,E1 -14775.044,E2 -14775.044} C_VEL
LIN {X 0,Y 334.266,Z 361.858,A -85,B 0,C 180,E1 -14776.305,E2 -14776.305} C_VEL
LIN {X 0,Y 331.954,Z 352.78,A -85,B 0,C 180,E1 -14777.688,E2 -14777.688} C_VEL
LIN {X 0,Y 329.852,Z 346.443,A -85,B 0,C 180,E1 -14778.64,E2 -14778.64} C_VEL
LIN {X 0,Y 328.508,Z 342.854,A -85,B 0,C 180,E1 -14779.19,E2 -14779.19} C_VEL
LIN {X 0,Y 329.297,Z 338.789,A -85,B 0,C 180,E1 -14782.593,E2 -14782.593} C_VEL
LIN {X 0,Y 330.412,Z 334.441,A -85,B 0,C 180,E1 -14786.701,E2 -14786.701} C_VEL
LIN {X 0,Y 331.236,Z 331.822,A -85,B 0,C 180,E1 -14789.551,E2 -14789.551} C_VEL
LIN {X 0,Y 331.771,Z 329.915,A -85,B 0,C 180,E1 -14792.077,E2 -14792.077} C_VEL
LIN {X 0,Y 331.994,Z 328.432,A -85,B 0,C 180,E1 -14794.861,E2 -14794.861} C_VEL
LIN {X 0,Y 332.118,Z 327.49,A -85,B 0,C 180,E1 -14797.857,E2 -14797.857} C_VEL
LIN {X 0,Y 332.264,Z 327.324,A -85,B 0,C 180,E1 -14800.975,E2 -14800.975} C_VEL
LIN {X 0,Y 332.585,Z 328.002,A -85,B 0,C 180,E1 -14804.215,E2 -14804.215} C_VEL
LIN {X 0,Y 333.085,Z 329.706,A -85,B 0,C 180,E1 -14807.531,E2 -14807.531} C_VEL
LIN {X 0,Y 333.776,Z 332.468,A -85,B 0,C 180,E1 -14810.825,E2 -14810.825} C_VEL
LIN {X 0,Y 334.611,Z 336.155,A -85,B 0,C 180,E1 -14813.978,E2 -14813.978} C_VEL
LIN {X 0,Y 335.509,Z 340.697,A -85,B 0,C 180,E1 -14817,E2 -14817} C_VEL
LIN {X 0,Y 335.66,Z 343.295,A -85,B 0,C 180,E1 -14818.436,E2 -14818.436} C_VEL
LIN {X 0,Y 334.222,Z 347.725,A -85,B 0,C 180,E1 -14820.386,E2 -14820.386} C_VEL
LIN {X 0,Y 331.372,Z 357.332,A -85,B 0,C 180,E1 -14824.229,E2 -14824.229} C_VEL
LIN {X 0,Y 330.49,Z 361.302,A -85,B 0,C 180,E1 -14825.727,E2 -14825.727} C_VEL
LIN {X 0,Y 333.478,Z 375.641,A -85,B 0,C 180,E1 -14826.989,E2 -14826.989} C_VEL
LIN {X 0,Y 334.807,Z 387.009,A -85,B 0,C 180,E1 -14828.057,E2 -14828.057} C_VEL
LIN {X 0,Y 334.703,Z 397.454,A -85,B 0,C 180,E1 -14829.086,E2 -14829.086} C_VEL
LIN {X 0,Y 333.678,Z 407.108,A -85,B 0,C 180,E1 -14830.146,E2 -14830.146} C_VEL
LIN {X 0,Y 331.727,Z 417.476,A -85,B 0,C 180,E1 -14831.47,E2 -14831.47} C_VEL
LIN {X 0,Y 329.943,Z 426.873,A -85,B 0,C 180,E1 -14832.969,E2 -14832.969} C_VEL
LIN {X 0,Y 328.255,Z 436.105,A -85,B 0,C 180,E1 -14834.794,E2 -14834.794} C_VEL
LIN {X 0,Y 327.006,Z 443.557,A -85,B 0,C 180,E1 -14836.642,E2 -14836.642} C_VEL
LIN {X 0,Y 325.845,Z 450.51,A -85,B 0,C 180,E1 -14838.807,E2 -14838.807} C_VEL
LIN {X 0,Y 325.395,Z 455.139,A -85,B 0,C 180,E1 -14840.678,E2 -14840.678} C_VEL
